REGION Network 1
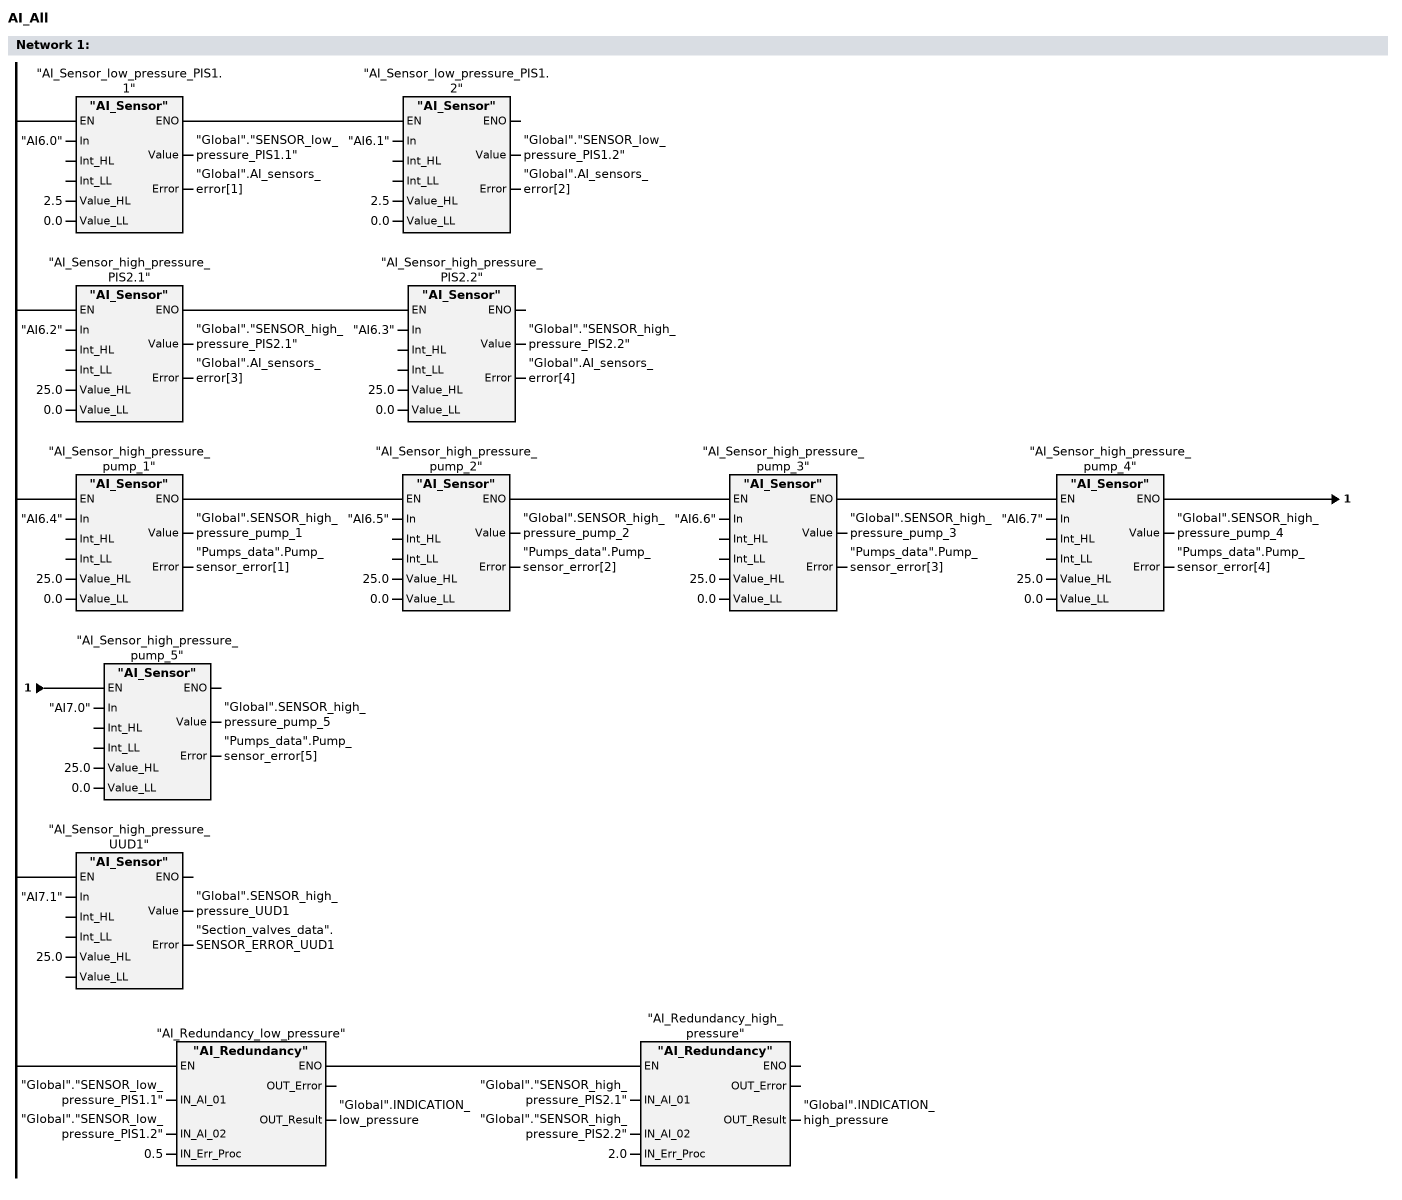
   RUNG wire#powerrail
      "AI_Sensor_low_pressure_PIS1.1"(In := "AI6.0", Int_HL :=, Int_LL :=, Value_HL := 2.5, Value_LL := 0.0, Value => "Global"."SENSOR_low_pressure_PIS1.1", Error => "Global".AI_sensors_error[1])
      "AI_Sensor_low_pressure_PIS1.2"(In := "AI6.1", Int_HL :=, Int_LL :=, Value_HL := 2.5, Value_LL := 0.0, Value => "Global"."SENSOR_low_pressure_PIS1.2", Error => "Global".AI_sensors_error[2])
   END_RUNG
   RUNG wire#powerrail
      "AI_Sensor_high_pressure_PIS2.1"(In := "AI6.2", Int_HL :=, Int_LL :=, Value_HL := 25.0, Value_LL := 0.0, Value => "Global"."SENSOR_high_pressure_PIS2.1", Error => "Global".AI_sensors_error[3])
      "AI_Sensor_high_pressure_PIS2.2"(In := "AI6.3", Int_HL :=, Int_LL :=, Value_HL := 25.0, Value_LL := 0.0, Value => "Global"."SENSOR_high_pressure_PIS2.2", Error => "Global".AI_sensors_error[4])
   END_RUNG
   RUNG wire#powerrail
      "AI_Sensor_high_pressure_pump_1"(In := "AI6.4", Int_HL :=, Int_LL :=, Value_HL := 25.0, Value_LL := 0.0, Value => "Global".SENSOR_high_pressure_pump_1, Error => "Pumps_data".Pump_sensor_error[1])
      "AI_Sensor_high_pressure_pump_2"(In := "AI6.5", Int_HL :=, Int_LL :=, Value_HL := 25.0, Value_LL := 0.0, Value => "Global".SENSOR_high_pressure_pump_2, Error => "Pumps_data".Pump_sensor_error[2])
      "AI_Sensor_high_pressure_pump_3"(In := "AI6.6", Int_HL :=, Int_LL :=, Value_HL := 25.0, Value_LL := 0.0, Value => "Global".SENSOR_high_pressure_pump_3, Error => "Pumps_data".Pump_sensor_error[3])
      "AI_Sensor_high_pressure_pump_4"(In := "AI6.7", Int_HL :=, Int_LL :=, Value_HL := 25.0, Value_LL := 0.0, Value => "Global".SENSOR_high_pressure_pump_4, Error => "Pumps_data".Pump_sensor_error[4])
      "AI_Sensor_high_pressure_pump_5"(In := "AI7.0", Int_HL :=, Int_LL :=, Value_HL := 25.0, Value_LL := 0.0, Value => "Global".SENSOR_high_pressure_pump_5, Error => "Pumps_data".Pump_sensor_error[5])
   END_RUNG
   RUNG wire#powerrail
      "AI_Sensor_high_pressure_UUD1"(In := "AI7.1", Int_HL :=, Int_LL :=, Value_HL := 25.0, Value_LL :=, Value => "Global".SENSOR_high_pressure_UUD1, Error => "Section_valves_data".SENSOR_ERROR_UUD1)
   END_RUNG
   RUNG wire#powerrail
      "AI_Redundancy_low_pressure"(IN_AI_01 := "Global"."SENSOR_low_pressure_PIS1.1", IN_AI_02 := "Global"."SENSOR_low_pressure_PIS1.2", IN_Err_Proc := 0.5, OUT_Error =>, OUT_Result => "Global".INDICATION_low_pressure)
      "AI_Redundancy_high_pressure"(IN_AI_01 := "Global"."SENSOR_high_pressure_PIS2.1", IN_AI_02 := "Global"."SENSOR_high_pressure_PIS2.2", IN_Err_Proc := 2.0, OUT_Error =>, OUT_Result => "Global".INDICATION_high_pressure)
   END_RUNG
   // the same network as SCL:
   "AI_Sensor_low_pressure_PIS1.1"(In := "AI6.0",   // "AI_Sensor"
                           Value_HL := 2.5,
                           Value_LL := 0.0,
                           Value => "Global"."SENSOR_low_pressure_PIS1.1",
                           Error => "Global".AI_sensors_error[1],
                           ENO => #_w1);
   IF #_w1 THEN
       "AI_Sensor_low_pressure_PIS1.2"(In := "AI6.1",   // "AI_Sensor"
                               Value_HL := 2.5,
                               Value_LL := 0.0,
                               Value => "Global"."SENSOR_low_pressure_PIS1.2",
                               Error => "Global".AI_sensors_error[2]);
   END_IF;
   "AI_Sensor_high_pressure_PIS2.1"(In := "AI6.2",   // "AI_Sensor"
                           Value_HL := 25.0,
                           Value_LL := 0.0,
                           Value => "Global"."SENSOR_high_pressure_PIS2.1",
                           Error => "Global".AI_sensors_error[3],
                           ENO => #_w2);
   IF #_w2 THEN
       "AI_Sensor_high_pressure_PIS2.2"(In := "AI6.3",   // "AI_Sensor"
                               Value_HL := 25.0,
                               Value_LL := 0.0,
                               Value => "Global"."SENSOR_high_pressure_PIS2.2",
                               Error => "Global".AI_sensors_error[4]);
   END_IF;
   "AI_Sensor_high_pressure_pump_1"(In := "AI6.4",   // "AI_Sensor"
                           Value_HL := 25.0,
                           Value_LL := 0.0,
                           Value => "Global".SENSOR_high_pressure_pump_1,
                           Error => "Pumps_data".Pump_sensor_error[1],
                           ENO => #_w3);
   "AI_Sensor_high_pressure_pump_2"(EN := #_w3,   // "AI_Sensor"
                           In := "AI6.5",
                           Value_HL := 25.0,
                           Value_LL := 0.0,
                           Value => "Global".SENSOR_high_pressure_pump_2,
                           Error => "Pumps_data".Pump_sensor_error[2],
                           ENO => #_w4);
   "AI_Sensor_high_pressure_pump_3"(EN := #_w4,   // "AI_Sensor"
                           In := "AI6.6",
                           Value_HL := 25.0,
                           Value_LL := 0.0,
                           Value => "Global".SENSOR_high_pressure_pump_3,
                           Error => "Pumps_data".Pump_sensor_error[3],
                           ENO => #_w5);
   "AI_Sensor_high_pressure_pump_4"(EN := #_w5,   // "AI_Sensor"
                           In := "AI6.7",
                           Value_HL := 25.0,
                           Value_LL := 0.0,
                           Value => "Global".SENSOR_high_pressure_pump_4,
                           Error => "Pumps_data".Pump_sensor_error[4],
                           ENO => #_w6);
   IF #_w6 THEN
       "AI_Sensor_high_pressure_pump_5"(In := "AI7.0",   // "AI_Sensor"
                               Value_HL := 25.0,
                               Value_LL := 0.0,
                               Value => "Global".SENSOR_high_pressure_pump_5,
                               Error => "Pumps_data".Pump_sensor_error[5]);
   END_IF;
   "AI_Sensor_high_pressure_UUD1"(In := "AI7.1",   // "AI_Sensor"
                           Value_HL := 25.0,
                           Value => "Global".SENSOR_high_pressure_UUD1,
                           Error => "Section_valves_data".SENSOR_ERROR_UUD1);
   "AI_Redundancy_low_pressure"(IN_AI_01 := "Global"."SENSOR_low_pressure_PIS1.1",   // "AI_Redundancy"
                           IN_AI_02 := "Global"."SENSOR_low_pressure_PIS1.2",
                           IN_Err_Proc := 0.5,
                           OUT_Result => "Global".INDICATION_low_pressure,
                           ENO => #_w7);
   IF #_w7 THEN
       "AI_Redundancy_high_pressure"(IN_AI_01 := "Global"."SENSOR_high_pressure_PIS2.1",   // "AI_Redundancy"
                               IN_AI_02 := "Global"."SENSOR_high_pressure_PIS2.2",
                               IN_Err_Proc := 2.0,
                               OUT_Result => "Global".INDICATION_high_pressure);
   END_IF;
END_REGION
END_FUNCTION

ORGANIZATION_BLOCK "Main"   // OB1, LAD, ProgramCycle
TITLE = "Main Program Sweep (Cycle)"
{ S7_Optimized_Access := 'TRUE' }
VERSION : 0.1
   VAR_INPUT
      Initial_Call : Bool;   // Initial call of this OB
      Remanence : Bool;   // =True, if remanent data are available
   END_VAR
   VAR_TEMP   // added for the SCL form of the ladder/FBD networks
      _w1 : Bool;
   END_VAR
BEGIN

REGION Network 1: Обработка входов
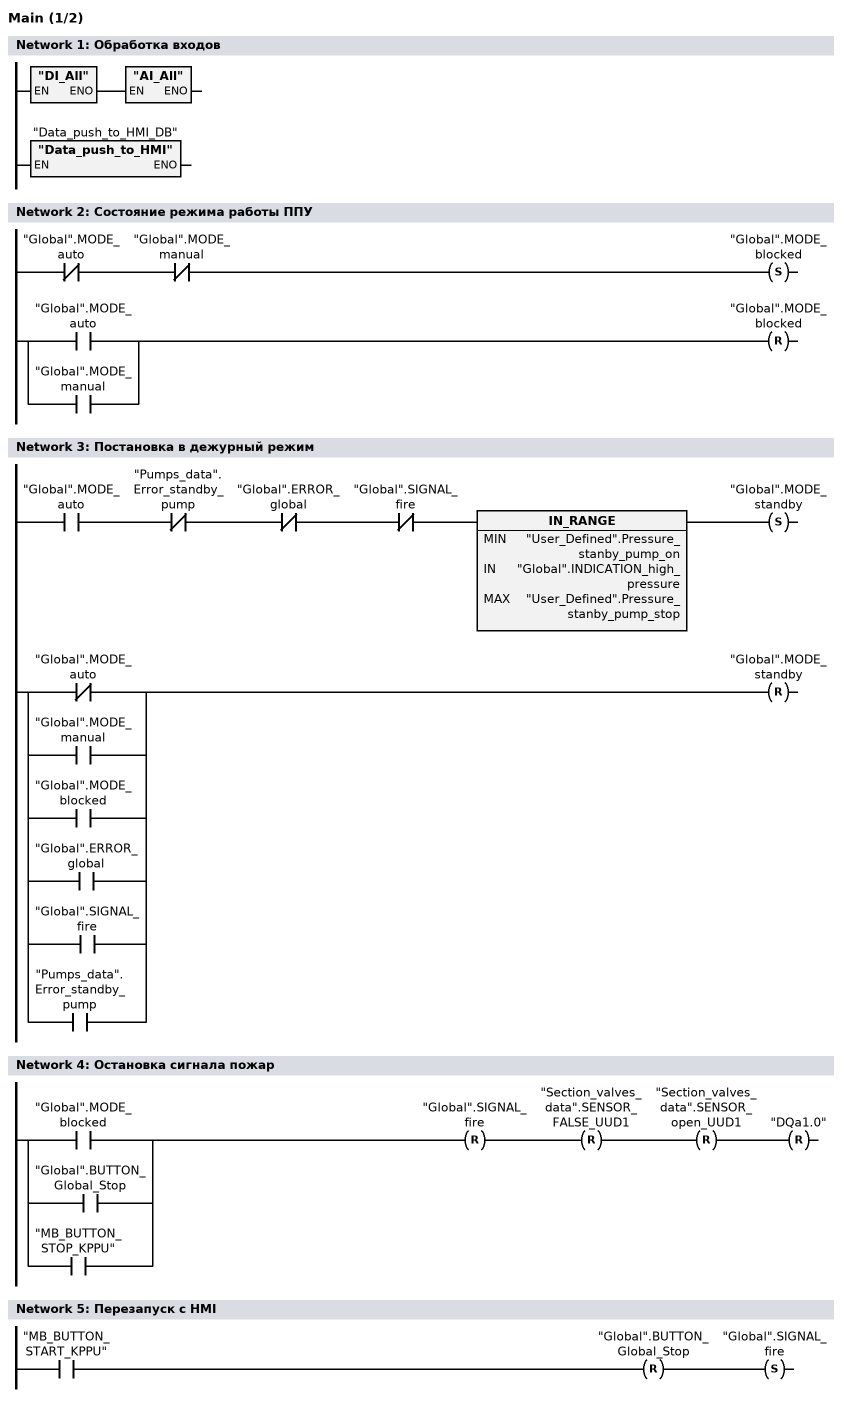
   RUNG wire#powerrail
      "DI_All"()
      "AI_All"()
   END_RUNG
   RUNG wire#powerrail
      "Data_push_to_HMI_DB"()
   END_RUNG
   // the same network as SCL:
   "DI_All"(ENO => #_w1);
   IF #_w1 THEN "AI_All"(); END_IF;
   "Data_push_to_HMI_DB"();   // "Data_push_to_HMI"
END_REGION

REGION Network 2: Состояние режима работы ППУ
   RUNG wire#powerrail
      I_Contact( "Global".MODE_auto )
      I_Contact( "Global".MODE_manual )
      S_Coil( "Global".MODE_blocked )
   END_RUNG
   RUNG wire#powerrail
      Contact( "Global".MODE_auto )
      wire#w1
      R_Coil( "Global".MODE_blocked )
   END_RUNG
   RUNG wire#powerrail
      Contact( "Global".MODE_manual )
   END_RUNG wire#w1
   // the same network as SCL:
   IF NOT "Global".MODE_auto AND NOT "Global".MODE_manual THEN "Global".MODE_blocked := TRUE; END_IF;
   IF "Global".MODE_auto OR "Global".MODE_manual THEN "Global".MODE_blocked := FALSE; END_IF;
END_REGION

REGION Network 3: Постановка в дежурный режим
   RUNG wire#powerrail
      Contact( "Global".MODE_auto )
      I_Contact( "Pumps_data".Error_standby_pump )
      I_Contact( "Global".ERROR_global )
      I_Contact( "Global".SIGNAL_fire )
      { S7_Templates := "SrcType := Real" } InRange(min := "User_Defined".Pressure_stanby_pump_on, in := "Global".INDICATION_high_pressure, max := "User_Defined".Pressure_stanby_pump_stop)
      S_Coil( "Global".MODE_standby )
   END_RUNG
   RUNG wire#powerrail
      I_Contact( "Global".MODE_auto )
      wire#w1
      R_Coil( "Global".MODE_standby )
   END_RUNG
   RUNG wire#powerrail
      Contact( "Global".MODE_manual )
   END_RUNG wire#w1
   RUNG wire#powerrail
      Contact( "Global".MODE_blocked )
   END_RUNG wire#w1
   RUNG wire#powerrail
      Contact( "Global".ERROR_global )
   END_RUNG wire#w1
   RUNG wire#powerrail
      Contact( "Global".SIGNAL_fire )
   END_RUNG wire#w1
   RUNG wire#powerrail
      Contact( "Pumps_data".Error_standby_pump )
   END_RUNG wire#w1
   // the same network as SCL:
   IF "Global".MODE_auto AND NOT "Pumps_data".Error_standby_pump AND NOT "Global".ERROR_global AND NOT "Global".SIGNAL_fire AND ("User_Defined".Pressure_stanby_pump_on <= "Global".INDICATION_high_pressure) AND ("Global".INDICATION_high_pressure <= "User_Defined".Pressure_stanby_pump_stop) THEN
       "Global".MODE_standby := TRUE;
   END_IF;
   IF NOT "Global".MODE_auto OR "Global".MODE_manual OR "Global".MODE_blocked OR "Global".ERROR_global OR "Global".SIGNAL_fire OR "Pumps_data".Error_standby_pump THEN
       "Global".MODE_standby := FALSE;
   END_IF;
END_REGION

REGION Network 4: Остановка сигнала пожар
   RUNG wire#powerrail
      Contact( "Global".MODE_blocked )
      wire#w1
      R_Coil( "Global".SIGNAL_fire )
      R_Coil( "Section_valves_data".SENSOR_FALSE_UUD1 )
      R_Coil( "Section_valves_data".SENSOR_open_UUD1 )
      R_Coil( "DQa1.0" )
   END_RUNG
   RUNG wire#powerrail
      Contact( "Global".BUTTON_Global_Stop )
   END_RUNG wire#w1
   RUNG wire#powerrail
      Contact( "MB_BUTTON_STOP_KPPU" )
   END_RUNG wire#w1
   // the same network as SCL:
   IF "Global".MODE_blocked OR "Global".BUTTON_Global_Stop OR "MB_BUTTON_STOP_KPPU" THEN
       "Global".SIGNAL_fire := FALSE;
       "Section_valves_data".SENSOR_FALSE_UUD1 := FALSE;
       "Section_valves_data".SENSOR_open_UUD1 := FALSE;
       "DQa1.0" := FALSE;
   END_IF;
END_REGION

REGION Network 5: Перезапуск с HMI
   RUNG wire#powerrail
      Contact( "MB_BUTTON_START_KPPU" )
      R_Coil( "Global".BUTTON_Global_Stop )
      S_Coil( "Global".SIGNAL_fire )
   END_RUNG
   // the same network as SCL:
   IF "MB_BUTTON_START_KPPU" THEN
       "Global".BUTTON_Global_Stop := FALSE;
       "Global".SIGNAL_fire := TRUE;
   END_IF;
END_REGION

REGION Network 6
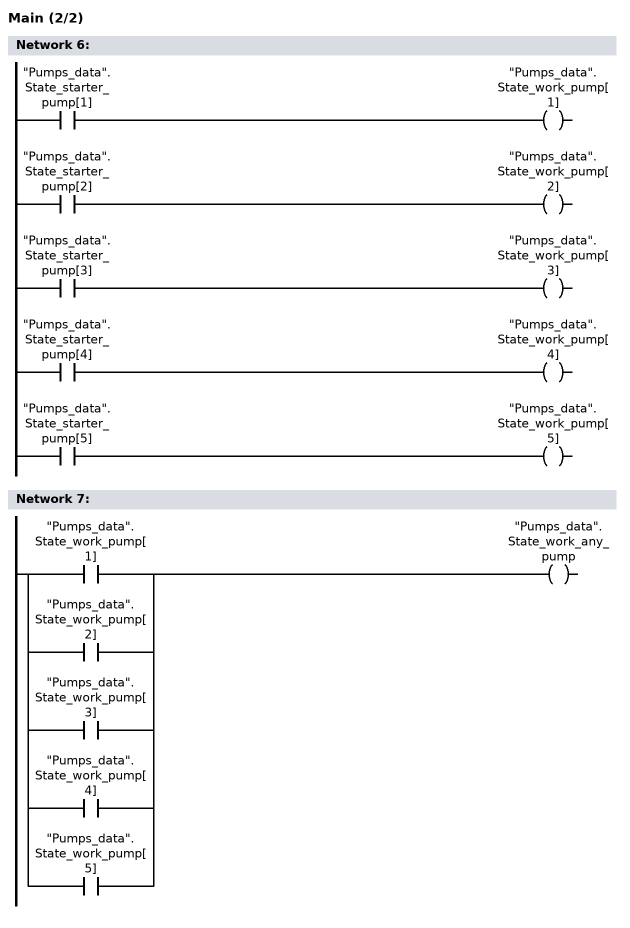
   RUNG wire#powerrail
      Contact( "Pumps_data".State_starter_pump[1] )
      Coil( "Pumps_data".State_work_pump[1] )
   END_RUNG
   RUNG wire#powerrail
      Contact( "Pumps_data".State_starter_pump[2] )
      Coil( "Pumps_data".State_work_pump[2] )
   END_RUNG
   RUNG wire#powerrail
      Contact( "Pumps_data".State_starter_pump[3] )
      Coil( "Pumps_data".State_work_pump[3] )
   END_RUNG
   RUNG wire#powerrail
      Contact( "Pumps_data".State_starter_pump[4] )
      Coil( "Pumps_data".State_work_pump[4] )
   END_RUNG
   RUNG wire#powerrail
      Contact( "Pumps_data".State_starter_pump[5] )
      Coil( "Pumps_data".State_work_pump[5] )
   END_RUNG
   // the same network as SCL:
   "Pumps_data".State_work_pump[1] := "Pumps_data".State_starter_pump[1];
   "Pumps_data".State_work_pump[2] := "Pumps_data".State_starter_pump[2];
   "Pumps_data".State_work_pump[3] := "Pumps_data".State_starter_pump[3];
   "Pumps_data".State_work_pump[4] := "Pumps_data".State_starter_pump[4];
   "Pumps_data".State_work_pump[5] := "Pumps_data".State_starter_pump[5];
END_REGION

REGION Network 7
   RUNG wire#powerrail
      Contact( "Pumps_data".State_work_pump[1] )
      wire#w1
      Coil( "Pumps_data".State_work_any_pump )
   END_RUNG
   RUNG wire#powerrail
      Contact( "Pumps_data".State_work_pump[2] )
   END_RUNG wire#w1
   RUNG wire#powerrail
      Contact( "Pumps_data".State_work_pump[3] )
   END_RUNG wire#w1
   RUNG wire#powerrail
      Contact( "Pumps_data".State_work_pump[4] )
   END_RUNG wire#w1
   RUNG wire#powerrail
      Contact( "Pumps_data".State_work_pump[5] )
   END_RUNG wire#w1
   // the same network as SCL:
   "Pumps_data".State_work_any_pump := "Pumps_data".State_work_pump[1] OR "Pumps_data".State_work_pump[2] OR "Pumps_data".State_work_pump[3] OR "Pumps_data".State_work_pump[4] OR "Pumps_data".State_work_pump[5];
END_REGION
END_ORGANIZATION_BLOCK

ORGANIZATION_BLOCK "Buttons"   // OB123, LAD, ProgramCycle
TITLE = "Main Program Sweep (Cycle)"
{ S7_Optimized_Access := 'TRUE' }
VERSION : 0.1
   VAR_INPUT
      Initial_Call : Bool;   // Initial call of this OB
      Remanence : Bool;   // =True, if remanent data are available
   END_VAR
   VAR_TEMP   // added for the SCL form of the ladder/FBD networks
      _w1 : Bool;
   END_VAR
BEGIN

REGION Network 1: Кнопка СТОП
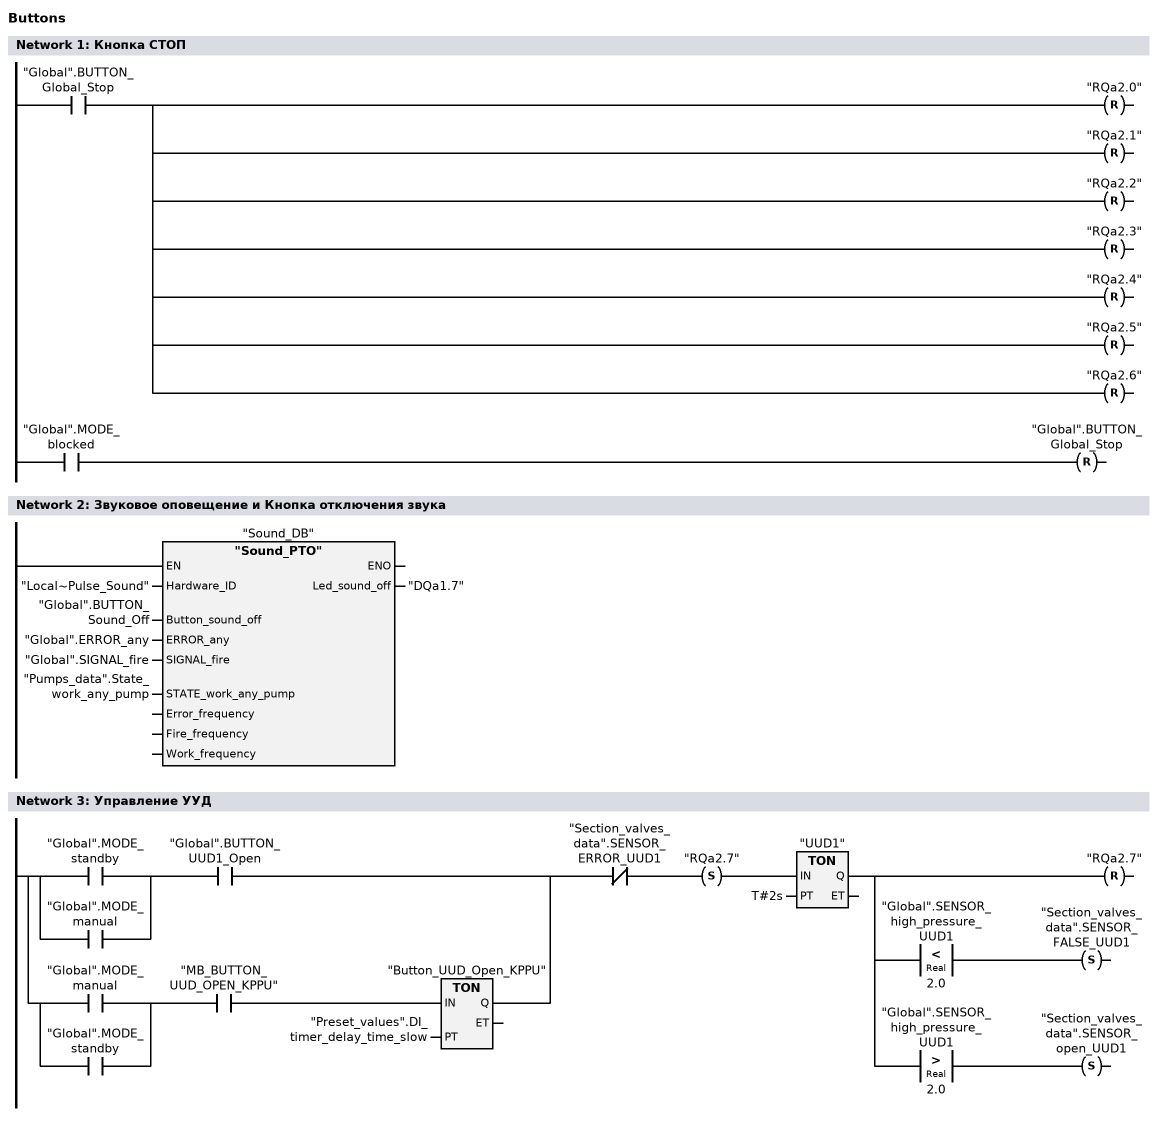
   RUNG wire#powerrail
      Contact( "Global".BUTTON_Global_Stop )
      wire#w1
      R_Coil( "RQa2.0" )
   END_RUNG
   RUNG wire#w1
      R_Coil( "RQa2.1" )
   END_RUNG
   RUNG wire#w1
      R_Coil( "RQa2.2" )
   END_RUNG
   RUNG wire#w1
      R_Coil( "RQa2.3" )
   END_RUNG
   RUNG wire#w1
      R_Coil( "RQa2.4" )
   END_RUNG
   RUNG wire#w1
      R_Coil( "RQa2.5" )
   END_RUNG
   RUNG wire#w1
      R_Coil( "RQa2.6" )
   END_RUNG
   RUNG wire#powerrail
      Contact( "Global".MODE_blocked )
      R_Coil( "Global".BUTTON_Global_Stop )
   END_RUNG
   // the same network as SCL:
   IF "Global".BUTTON_Global_Stop THEN
       "RQa2.0" := FALSE;
       "RQa2.1" := FALSE;
       "RQa2.2" := FALSE;
       "RQa2.3" := FALSE;
       "RQa2.4" := FALSE;
       "RQa2.5" := FALSE;
       "RQa2.6" := FALSE;
   END_IF;
   IF "Global".MODE_blocked THEN "Global".BUTTON_Global_Stop := FALSE; END_IF;
END_REGION

REGION Network 2: Звуковое оповещение и Кнопка отключения звука
   RUNG wire#powerrail
      "Sound_DB"(Hardware_ID := "Local~Pulse_Sound", Button_sound_off := "Global".BUTTON_Sound_Off, ERROR_any := "Global".ERROR_any, SIGNAL_fire := "Global".SIGNAL_fire, STATE_work_any_pump := "Pumps_data".State_work_any_pump, Error_frequency :=, Fire_frequency :=, Work_frequency :=, Led_sound_off => "DQa1.7")
   END_RUNG
   // the same network as SCL:
   "Sound_DB"(Hardware_ID := "Local~Pulse_Sound",   // "Sound_PTO"
              Button_sound_off := "Global".BUTTON_Sound_Off,
              ERROR_any := "Global".ERROR_any,
              SIGNAL_fire := "Global".SIGNAL_fire,
              STATE_work_any_pump := "Pumps_data".State_work_any_pump,
              Led_sound_off => "DQa1.7");
END_REGION

REGION Network 3: Управление УУД
   "Button_UUD_Open_KPPU".TON(IN := ("Global".MODE_manual OR "Global".MODE_standby) AND "MB_BUTTON_UUD_OPEN_KPPU",
                           PT := "Preset_values".DI_timer_delay_time_slow);
   #_w1 := ((("Global".MODE_standby OR "Global".MODE_manual) AND "Global".BUTTON_UUD1_Open) OR "Button_UUD_Open_KPPU".Q) AND NOT "Section_valves_data".SENSOR_ERROR_UUD1;
   IF #_w1 THEN "RQa2.7" := TRUE; END_IF;
   "UUD1".TON(IN := #_w1, PT := T#2s);
   IF "UUD1".Q THEN "RQa2.7" := FALSE; END_IF;
   IF "UUD1".Q AND ("Global".SENSOR_high_pressure_UUD1 < 2.0) THEN
       "Section_valves_data".SENSOR_FALSE_UUD1 := TRUE;
   END_IF;
   IF "UUD1".Q AND ("Global".SENSOR_high_pressure_UUD1 > 2.0) THEN
       "Section_valves_data".SENSOR_open_UUD1 := TRUE;
   END_IF;
END_REGION
END_ORGANIZATION_BLOCK

ORGANIZATION_BLOCK "Errors"   // OB124, LAD, ProgramCycle
TITLE = "Main Program Sweep (Cycle)"
{ S7_Optimized_Access := 'TRUE' }
VERSION : 0.1
   VAR_INPUT
      Initial_Call : Bool;   // Initial call of this OB
      Remanence : Bool;   // =True, if remanent data are available
   END_VAR
   VAR_TEMP   // added for the SCL form of the ladder/FBD networks
      _w1 : Bool;
      _w2 : Bool;
      _w3 : Bool;
      _w4 : Bool;
   END_VAR
BEGIN

REGION Network 1: Нет воды
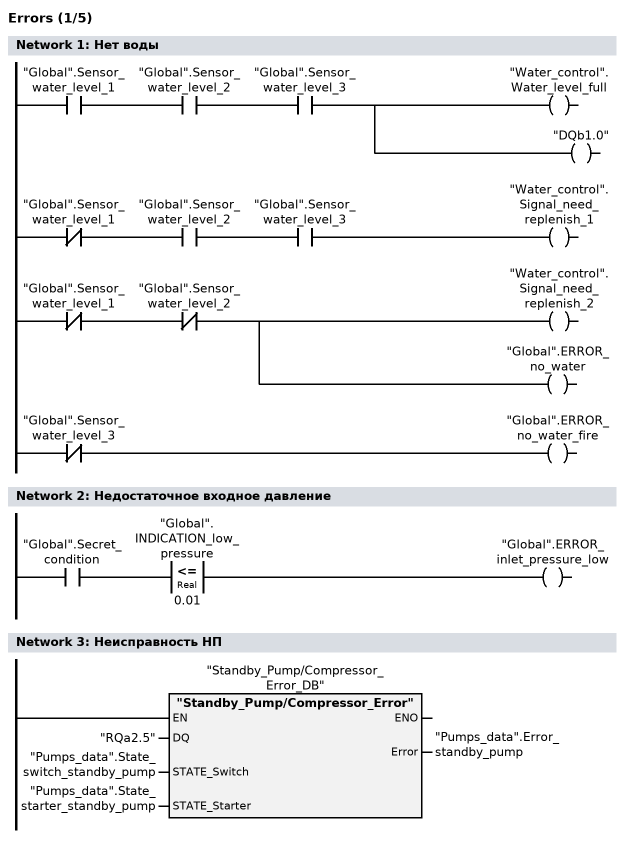
   RUNG wire#powerrail
      Contact( "Global".Sensor_water_level_1 )
      Contact( "Global".Sensor_water_level_2 )
      Contact( "Global".Sensor_water_level_3 )
      wire#w1
      Coil( "Water_control".Water_level_full )
   END_RUNG
   RUNG wire#w1
      Coil( "DQb1.0" )
   END_RUNG
   RUNG wire#powerrail
      I_Contact( "Global".Sensor_water_level_1 )
      Contact( "Global".Sensor_water_level_2 )
      Contact( "Global".Sensor_water_level_3 )
      Coil( "Water_control".Signal_need_replenish_1 )
   END_RUNG
   RUNG wire#powerrail
      I_Contact( "Global".Sensor_water_level_1 )
      I_Contact( "Global".Sensor_water_level_2 )
      wire#w2
      Coil( "Water_control".Signal_need_replenish_2 )
   END_RUNG
   RUNG wire#w2
      Coil( "Global".ERROR_no_water )
   END_RUNG
   RUNG wire#powerrail
      I_Contact( "Global".Sensor_water_level_3 )
      Coil( "Global".ERROR_no_water_fire )
   END_RUNG
   // the same network as SCL:
   "Water_control".Water_level_full := "Global".Sensor_water_level_1 AND "Global".Sensor_water_level_2 AND "Global".Sensor_water_level_3;
   "DQb1.0" := "Water_control".Water_level_full;
   "Water_control".Signal_need_replenish_1 := NOT "Global".Sensor_water_level_1 AND "Global".Sensor_water_level_2 AND "Global".Sensor_water_level_3;
   "Water_control".Signal_need_replenish_2 := NOT "Global".Sensor_water_level_1 AND NOT "Global".Sensor_water_level_2;
   "Global".ERROR_no_water := "Water_control".Signal_need_replenish_2;
   "Global".ERROR_no_water_fire := NOT "Global".Sensor_water_level_3;
END_REGION

REGION Network 2: Недостаточное входное давление
   RUNG wire#powerrail
      Contact( "Global".Secret_condition )
      { S7_Templates := "SrcType := Real" } LE_Contact(in1 := "Global".INDICATION_low_pressure, in2 := 0.01)
      Coil( "Global".ERROR_inlet_pressure_low )
   END_RUNG
   // the same network as SCL:
   "Global".ERROR_inlet_pressure_low := "Global".Secret_condition AND ("Global".INDICATION_low_pressure <= 0.01);
END_REGION

REGION Network 3: Неисправность НП
   RUNG wire#powerrail
      "Standby_Pump/Compressor_Error_DB"(DQ := "RQa2.5", STATE_Switch := "Pumps_data".State_switch_standby_pump, STATE_Starter := "Pumps_data".State_starter_standby_pump, Error => "Pumps_data".Error_standby_pump)
   END_RUNG
   // the same network as SCL:
   "Standby_Pump/Compressor_Error_DB"(DQ := "RQa2.5",   // "Standby_Pump/Compressor_Error"
                           STATE_Switch := "Pumps_data".State_switch_standby_pump,
                           STATE_Starter := "Pumps_data".State_starter_standby_pump,
                           Error => "Pumps_data".Error_standby_pump);
END_REGION

REGION Network 4: Неисправности НБ
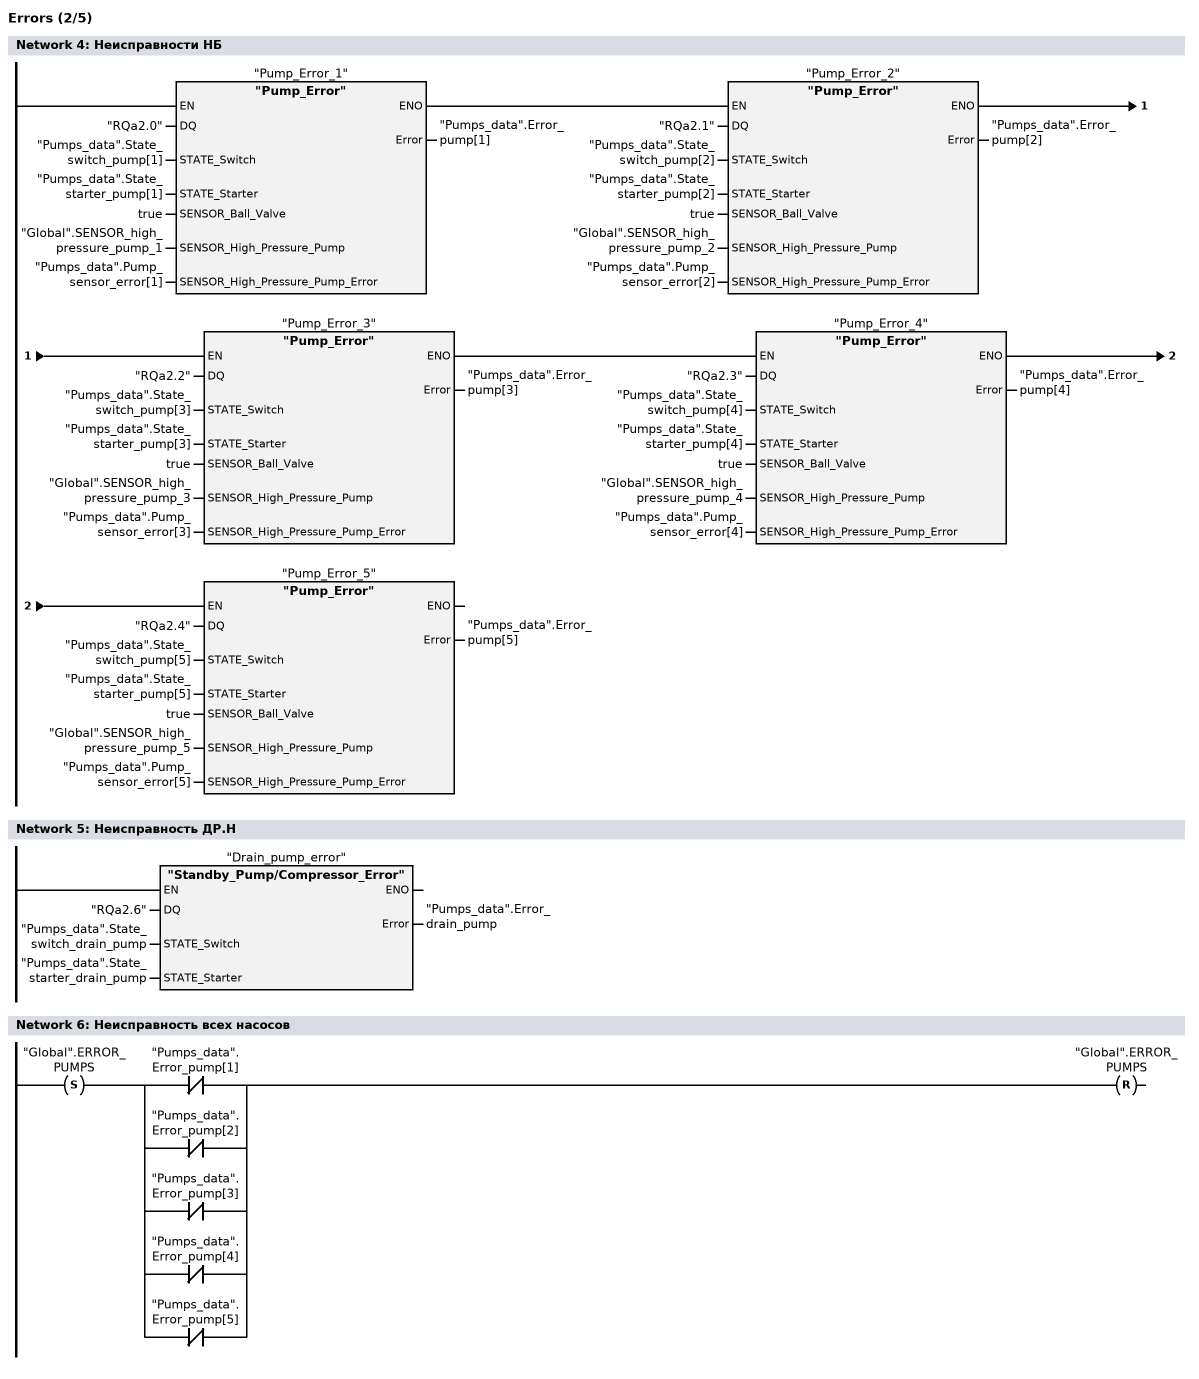
   RUNG wire#powerrail
      "Pump_Error_1"(DQ := "RQa2.0", STATE_Switch := "Pumps_data".State_switch_pump[1], STATE_Starter := "Pumps_data".State_starter_pump[1], SENSOR_Ball_Valve := true, SENSOR_High_Pressure_Pump := "Global".SENSOR_high_pressure_pump_1, SENSOR_High_Pressure_Pump_Error := "Pumps_data".Pump_sensor_error[1], Error => "Pumps_data".Error_pump[1])
      "Pump_Error_2"(DQ := "RQa2.1", STATE_Switch := "Pumps_data".State_switch_pump[2], STATE_Starter := "Pumps_data".State_starter_pump[2], SENSOR_Ball_Valve := true, SENSOR_High_Pressure_Pump := "Global".SENSOR_high_pressure_pump_2, SENSOR_High_Pressure_Pump_Error := "Pumps_data".Pump_sensor_error[2], Error => "Pumps_data".Error_pump[2])
      "Pump_Error_3"(DQ := "RQa2.2", STATE_Switch := "Pumps_data".State_switch_pump[3], STATE_Starter := "Pumps_data".State_starter_pump[3], SENSOR_Ball_Valve := true, SENSOR_High_Pressure_Pump := "Global".SENSOR_high_pressure_pump_3, SENSOR_High_Pressure_Pump_Error := "Pumps_data".Pump_sensor_error[3], Error => "Pumps_data".Error_pump[3])
      "Pump_Error_4"(DQ := "RQa2.3", STATE_Switch := "Pumps_data".State_switch_pump[4], STATE_Starter := "Pumps_data".State_starter_pump[4], SENSOR_Ball_Valve := true, SENSOR_High_Pressure_Pump := "Global".SENSOR_high_pressure_pump_4, SENSOR_High_Pressure_Pump_Error := "Pumps_data".Pump_sensor_error[4], Error => "Pumps_data".Error_pump[4])
      "Pump_Error_5"(DQ := "RQa2.4", STATE_Switch := "Pumps_data".State_switch_pump[5], STATE_Starter := "Pumps_data".State_starter_pump[5], SENSOR_Ball_Valve := true, SENSOR_High_Pressure_Pump := "Global".SENSOR_high_pressure_pump_5, SENSOR_High_Pressure_Pump_Error := "Pumps_data".Pump_sensor_error[5], Error => "Pumps_data".Error_pump[5])
   END_RUNG
   // the same network as SCL:
   "Pump_Error_1"(DQ := "RQa2.0",   // "Pump_Error"
                  STATE_Switch := "Pumps_data".State_switch_pump[1],
                  STATE_Starter := "Pumps_data".State_starter_pump[1],
                  SENSOR_Ball_Valve := true,
                  SENSOR_High_Pressure_Pump := "Global".SENSOR_high_pressure_pump_1,
                  SENSOR_High_Pressure_Pump_Error := "Pumps_data".Pump_sensor_error[1],
                  Error => "Pumps_data".Error_pump[1],
                  ENO => #_w1);
   "Pump_Error_2"(EN := #_w1,   // "Pump_Error"
                  DQ := "RQa2.1",
                  STATE_Switch := "Pumps_data".State_switch_pump[2],
                  STATE_Starter := "Pumps_data".State_starter_pump[2],
                  SENSOR_Ball_Valve := true,
                  SENSOR_High_Pressure_Pump := "Global".SENSOR_high_pressure_pump_2,
                  SENSOR_High_Pressure_Pump_Error := "Pumps_data".Pump_sensor_error[2],
                  Error => "Pumps_data".Error_pump[2],
                  ENO => #_w2);
   "Pump_Error_3"(EN := #_w2,   // "Pump_Error"
                  DQ := "RQa2.2",
                  STATE_Switch := "Pumps_data".State_switch_pump[3],
                  STATE_Starter := "Pumps_data".State_starter_pump[3],
                  SENSOR_Ball_Valve := true,
                  SENSOR_High_Pressure_Pump := "Global".SENSOR_high_pressure_pump_3,
                  SENSOR_High_Pressure_Pump_Error := "Pumps_data".Pump_sensor_error[3],
                  Error => "Pumps_data".Error_pump[3],
                  ENO => #_w3);
   "Pump_Error_4"(EN := #_w3,   // "Pump_Error"
                  DQ := "RQa2.3",
                  STATE_Switch := "Pumps_data".State_switch_pump[4],
                  STATE_Starter := "Pumps_data".State_starter_pump[4],
                  SENSOR_Ball_Valve := true,
                  SENSOR_High_Pressure_Pump := "Global".SENSOR_high_pressure_pump_4,
                  SENSOR_High_Pressure_Pump_Error := "Pumps_data".Pump_sensor_error[4],
                  Error => "Pumps_data".Error_pump[4],
                  ENO => #_w4);
   IF #_w4 THEN
       "Pump_Error_5"(DQ := "RQa2.4",   // "Pump_Error"
                      STATE_Switch := "Pumps_data".State_switch_pump[5],
                      STATE_Starter := "Pumps_data".State_starter_pump[5],
                      SENSOR_Ball_Valve := true,
                      SENSOR_High_Pressure_Pump := "Global".SENSOR_high_pressure_pump_5,
                      SENSOR_High_Pressure_Pump_Error := "Pumps_data".Pump_sensor_error[5],
                      Error => "Pumps_data".Error_pump[5]);
   END_IF;
END_REGION

REGION Network 5: Неисправность ДР.Н
   RUNG wire#powerrail
      "Drain_pump_error"(DQ := "RQa2.6", STATE_Switch := "Pumps_data".State_switch_drain_pump, STATE_Starter := "Pumps_data".State_starter_drain_pump, Error => "Pumps_data".Error_drain_pump)
   END_RUNG
   // the same network as SCL:
   "Drain_pump_error"(DQ := "RQa2.6",   // "Standby_Pump/Compressor_Error"
                      STATE_Switch := "Pumps_data".State_switch_drain_pump,
                      STATE_Starter := "Pumps_data".State_starter_drain_pump,
                      Error => "Pumps_data".Error_drain_pump);
END_REGION

REGION Network 6: Неисправность всех насосов
   RUNG wire#powerrail
      S_Coil( "Global".ERROR_PUMPS )
      wire#w1
      I_Contact( "Pumps_data".Error_pump[1] )
      wire#w2
      R_Coil( "Global".ERROR_PUMPS )
   END_RUNG
   RUNG wire#w1
      I_Contact( "Pumps_data".Error_pump[2] )
   END_RUNG wire#w2
   RUNG wire#w1
      I_Contact( "Pumps_data".Error_pump[3] )
   END_RUNG wire#w2
   RUNG wire#w1
      I_Contact( "Pumps_data".Error_pump[4] )
   END_RUNG wire#w2
   RUNG wire#w1
      I_Contact( "Pumps_data".Error_pump[5] )
   END_RUNG wire#w2
   // the same network as SCL:
   "Global".ERROR_PUMPS := TRUE;
   IF NOT "Pumps_data".Error_pump[1] OR NOT "Pumps_data".Error_pump[2] OR NOT "Pumps_data".Error_pump[3] OR NOT "Pumps_data".Error_pump[4] OR NOT "Pumps_data".Error_pump[5] THEN
       "Global".ERROR_PUMPS := FALSE;
   END_IF;
END_REGION

REGION Network 7: Неисправность любого насоса кроме резервного
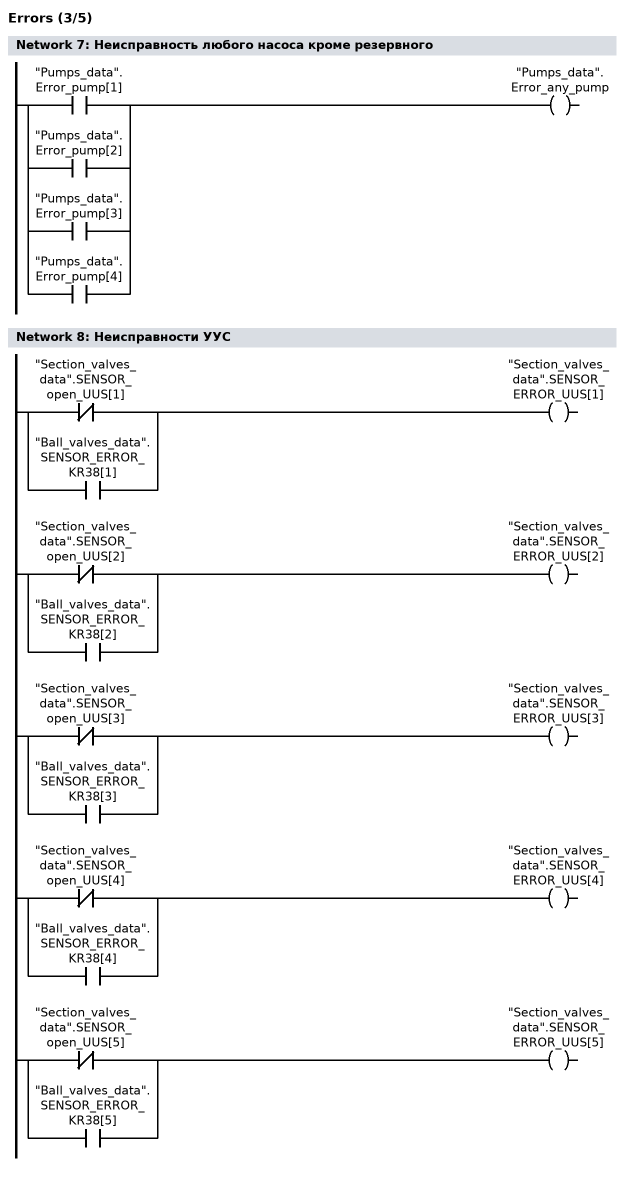
   RUNG wire#powerrail
      Contact( "Pumps_data".Error_pump[1] )
      wire#w1
      Coil( "Pumps_data".Error_any_pump )
   END_RUNG
   RUNG wire#powerrail
      Contact( "Pumps_data".Error_pump[2] )
   END_RUNG wire#w1
   RUNG wire#powerrail
      Contact( "Pumps_data".Error_pump[3] )
   END_RUNG wire#w1
   RUNG wire#powerrail
      Contact( "Pumps_data".Error_pump[4] )
   END_RUNG wire#w1
   // the same network as SCL:
   "Pumps_data".Error_any_pump := "Pumps_data".Error_pump[1] OR "Pumps_data".Error_pump[2] OR "Pumps_data".Error_pump[3] OR "Pumps_data".Error_pump[4];
END_REGION

REGION Network 8: Неисправности УУС
   RUNG wire#powerrail
      I_Contact( "Section_valves_data".SENSOR_open_UUS[1] )
      wire#w1
      Coil( "Section_valves_data".SENSOR_ERROR_UUS[1] )
   END_RUNG
   RUNG wire#powerrail
      Contact( "Ball_valves_data".SENSOR_ERROR_KR38[1] )
   END_RUNG wire#w1
   RUNG wire#powerrail
      I_Contact( "Section_valves_data".SENSOR_open_UUS[2] )
      wire#w2
      Coil( "Section_valves_data".SENSOR_ERROR_UUS[2] )
   END_RUNG
   RUNG wire#powerrail
      Contact( "Ball_valves_data".SENSOR_ERROR_KR38[2] )
   END_RUNG wire#w2
   RUNG wire#powerrail
      I_Contact( "Section_valves_data".SENSOR_open_UUS[3] )
      wire#w3
      Coil( "Section_valves_data".SENSOR_ERROR_UUS[3] )
   END_RUNG
   RUNG wire#powerrail
      Contact( "Ball_valves_data".SENSOR_ERROR_KR38[3] )
   END_RUNG wire#w3
   RUNG wire#powerrail
      I_Contact( "Section_valves_data".SENSOR_open_UUS[4] )
      wire#w4
      Coil( "Section_valves_data".SENSOR_ERROR_UUS[4] )
   END_RUNG
   RUNG wire#powerrail
      Contact( "Ball_valves_data".SENSOR_ERROR_KR38[4] )
   END_RUNG wire#w4
   RUNG wire#powerrail
      I_Contact( "Section_valves_data".SENSOR_open_UUS[5] )
      wire#w5
      Coil( "Section_valves_data".SENSOR_ERROR_UUS[5] )
   END_RUNG
   RUNG wire#powerrail
      Contact( "Ball_valves_data".SENSOR_ERROR_KR38[5] )
   END_RUNG wire#w5
   // the same network as SCL:
   "Section_valves_data".SENSOR_ERROR_UUS[1] := NOT "Section_valves_data".SENSOR_open_UUS[1] OR "Ball_valves_data".SENSOR_ERROR_KR38[1];
   "Section_valves_data".SENSOR_ERROR_UUS[2] := NOT "Section_valves_data".SENSOR_open_UUS[2] OR "Ball_valves_data".SENSOR_ERROR_KR38[2];
   "Section_valves_data".SENSOR_ERROR_UUS[3] := NOT "Section_valves_data".SENSOR_open_UUS[3] OR "Ball_valves_data".SENSOR_ERROR_KR38[3];
   "Section_valves_data".SENSOR_ERROR_UUS[4] := NOT "Section_valves_data".SENSOR_open_UUS[4] OR "Ball_valves_data".SENSOR_ERROR_KR38[4];
   "Section_valves_data".SENSOR_ERROR_UUS[5] := NOT "Section_valves_data".SENSOR_open_UUS[5] OR "Ball_valves_data".SENSOR_ERROR_KR38[5];
END_REGION

REGION Network 9: Неисправность всех УУС - все закрыты
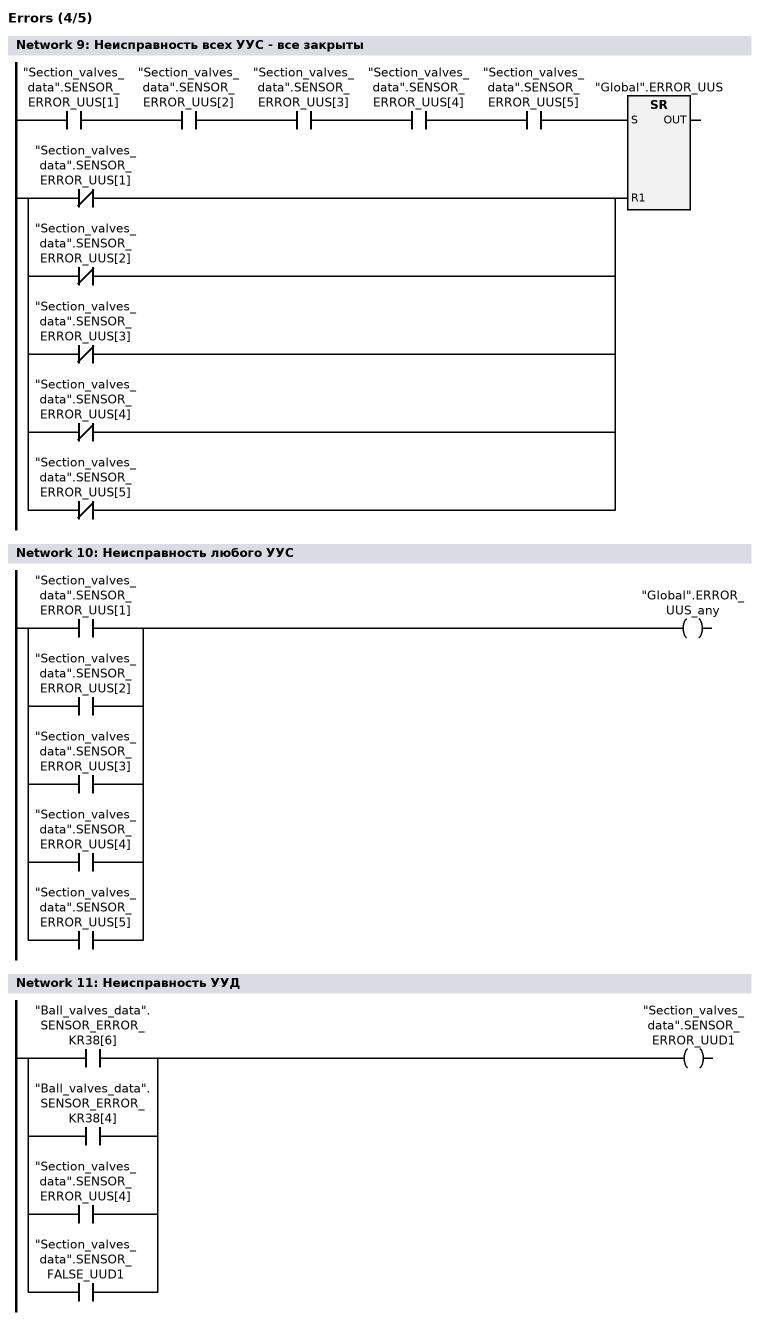
   RUNG wire#powerrail
      Contact( "Section_valves_data".SENSOR_ERROR_UUS[1] )
      Contact( "Section_valves_data".SENSOR_ERROR_UUS[2] )
      Contact( "Section_valves_data".SENSOR_ERROR_UUS[3] )
      Contact( "Section_valves_data".SENSOR_ERROR_UUS[4] )
      Contact( "Section_valves_data".SENSOR_ERROR_UUS[5] )
      S_SR(operand := "Global".ERROR_UUS, r1 := wire#w1)
   END_RUNG
   RUNG wire#powerrail
      I_Contact( "Section_valves_data".SENSOR_ERROR_UUS[1] )
   END_RUNG wire#w1
   RUNG wire#powerrail
      I_Contact( "Section_valves_data".SENSOR_ERROR_UUS[2] )
   END_RUNG wire#w1
   RUNG wire#powerrail
      I_Contact( "Section_valves_data".SENSOR_ERROR_UUS[3] )
   END_RUNG wire#w1
   RUNG wire#powerrail
      I_Contact( "Section_valves_data".SENSOR_ERROR_UUS[4] )
   END_RUNG wire#w1
   RUNG wire#powerrail
      I_Contact( "Section_valves_data".SENSOR_ERROR_UUS[5] )
   END_RUNG wire#w1
   // the same network as SCL:
   IF "Section_valves_data".SENSOR_ERROR_UUS[1] AND "Section_valves_data".SENSOR_ERROR_UUS[2] AND "Section_valves_data".SENSOR_ERROR_UUS[3] AND "Section_valves_data".SENSOR_ERROR_UUS[4] AND "Section_valves_data".SENSOR_ERROR_UUS[5] THEN
       "Global".ERROR_UUS := TRUE;   // SR flip-flop
   END_IF;
   IF NOT "Section_valves_data".SENSOR_ERROR_UUS[1] OR NOT "Section_valves_data".SENSOR_ERROR_UUS[2] OR NOT "Section_valves_data".SENSOR_ERROR_UUS[3] OR NOT "Section_valves_data".SENSOR_ERROR_UUS[4] OR NOT "Section_valves_data".SENSOR_ERROR_UUS[5] THEN
       "Global".ERROR_UUS := FALSE;
   END_IF;
END_REGION

REGION Network 10: Неисправность любого УУС
   RUNG wire#powerrail
      Contact( "Section_valves_data".SENSOR_ERROR_UUS[1] )
      wire#w1
      Coil( "Global".ERROR_UUS_any )
   END_RUNG
   RUNG wire#powerrail
      Contact( "Section_valves_data".SENSOR_ERROR_UUS[2] )
   END_RUNG wire#w1
   RUNG wire#powerrail
      Contact( "Section_valves_data".SENSOR_ERROR_UUS[3] )
   END_RUNG wire#w1
   RUNG wire#powerrail
      Contact( "Section_valves_data".SENSOR_ERROR_UUS[4] )
   END_RUNG wire#w1
   RUNG wire#powerrail
      Contact( "Section_valves_data".SENSOR_ERROR_UUS[5] )
   END_RUNG wire#w1
   // the same network as SCL:
   "Global".ERROR_UUS_any := "Section_valves_data".SENSOR_ERROR_UUS[1] OR "Section_valves_data".SENSOR_ERROR_UUS[2] OR "Section_valves_data".SENSOR_ERROR_UUS[3] OR "Section_valves_data".SENSOR_ERROR_UUS[4] OR "Section_valves_data".SENSOR_ERROR_UUS[5];
END_REGION

REGION Network 11: Неисправность УУД
   RUNG wire#powerrail
      Contact( "Ball_valves_data".SENSOR_ERROR_KR38[6] )
      wire#w1
      Coil( "Section_valves_data".SENSOR_ERROR_UUD1 )
   END_RUNG
   RUNG wire#powerrail
      Contact( "Ball_valves_data".SENSOR_ERROR_KR38[4] )
   END_RUNG wire#w1
   RUNG wire#powerrail
      Contact( "Section_valves_data".SENSOR_ERROR_UUS[4] )
   END_RUNG wire#w1
   RUNG wire#powerrail
      Contact( "Section_valves_data".SENSOR_FALSE_UUD1 )
   END_RUNG wire#w1
   // the same network as SCL:
   "Section_valves_data".SENSOR_ERROR_UUD1 := "Ball_valves_data".SENSOR_ERROR_KR38[6] OR "Ball_valves_data".SENSOR_ERROR_KR38[4] OR "Section_valves_data".SENSOR_ERROR_UUS[4] OR "Section_valves_data".SENSOR_FALSE_UUD1;
END_REGION

REGION Network 12: Неисправность любого шарового крана
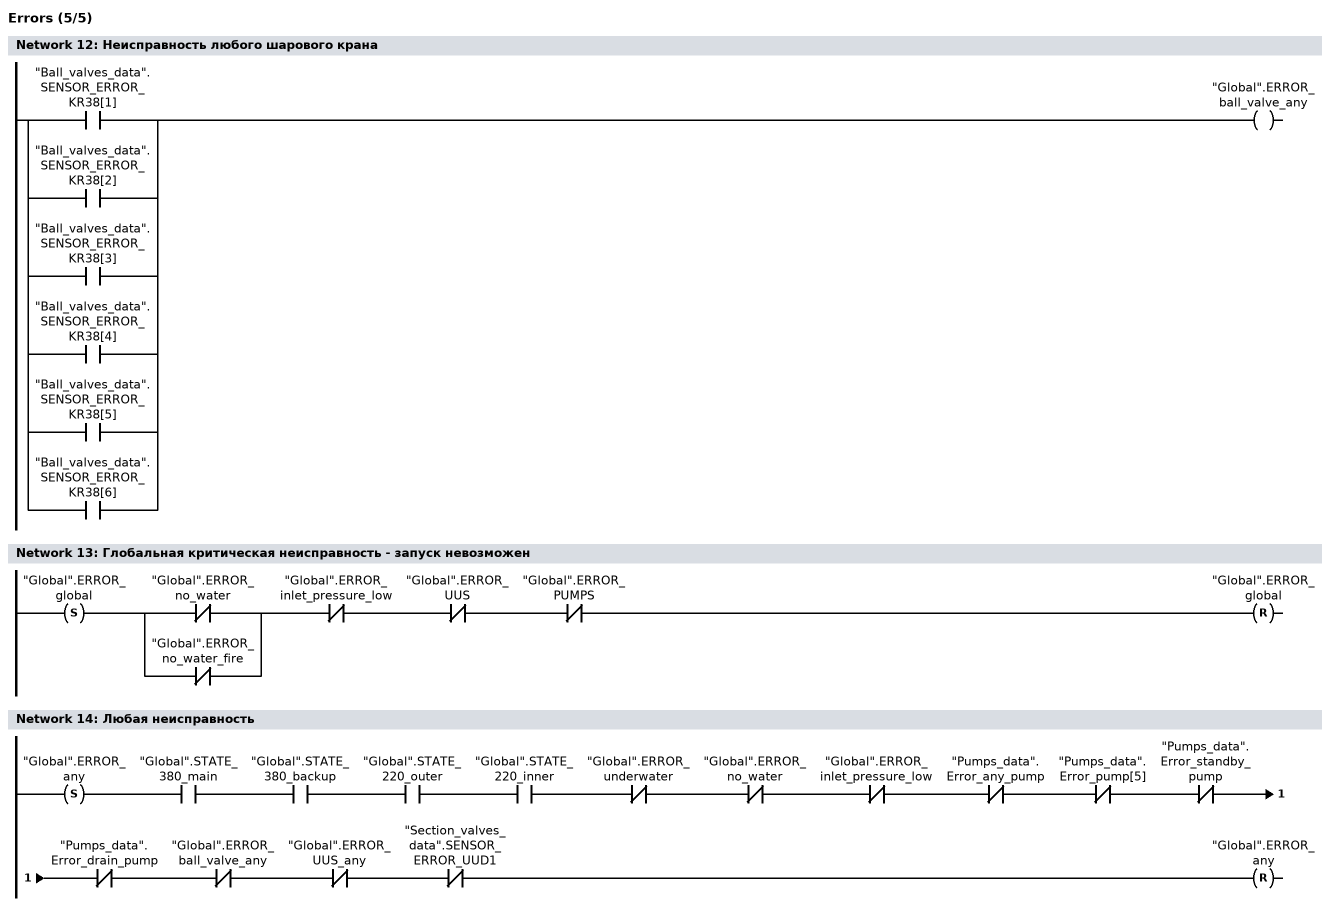
   RUNG wire#powerrail
      Contact( "Ball_valves_data".SENSOR_ERROR_KR38[1] )
      wire#w1
      Coil( "Global".ERROR_ball_valve_any )
   END_RUNG
   RUNG wire#powerrail
      Contact( "Ball_valves_data".SENSOR_ERROR_KR38[2] )
   END_RUNG wire#w1
   RUNG wire#powerrail
      Contact( "Ball_valves_data".SENSOR_ERROR_KR38[3] )
   END_RUNG wire#w1
   RUNG wire#powerrail
      Contact( "Ball_valves_data".SENSOR_ERROR_KR38[4] )
   END_RUNG wire#w1
   RUNG wire#powerrail
      Contact( "Ball_valves_data".SENSOR_ERROR_KR38[5] )
   END_RUNG wire#w1
   RUNG wire#powerrail
      Contact( "Ball_valves_data".SENSOR_ERROR_KR38[6] )
   END_RUNG wire#w1
   // the same network as SCL:
   "Global".ERROR_ball_valve_any := "Ball_valves_data".SENSOR_ERROR_KR38[1] OR "Ball_valves_data".SENSOR_ERROR_KR38[2] OR "Ball_valves_data".SENSOR_ERROR_KR38[3] OR "Ball_valves_data".SENSOR_ERROR_KR38[4] OR "Ball_valves_data".SENSOR_ERROR_KR38[5] OR "Ball_valves_data".SENSOR_ERROR_KR38[6];
END_REGION

REGION Network 13: Глобальная критическая неисправность - запуск невозможен
   RUNG wire#powerrail
      S_Coil( "Global".ERROR_global )
      wire#w1
      I_Contact( "Global".ERROR_no_water )
      wire#w2
      I_Contact( "Global".ERROR_inlet_pressure_low )
      I_Contact( "Global".ERROR_UUS )
      I_Contact( "Global".ERROR_PUMPS )
      R_Coil( "Global".ERROR_global )
   END_RUNG
   RUNG wire#w1
      I_Contact( "Global".ERROR_no_water_fire )
   END_RUNG wire#w2
   // the same network as SCL:
   "Global".ERROR_global := TRUE;
   IF (NOT "Global".ERROR_no_water OR NOT "Global".ERROR_no_water_fire) AND NOT "Global".ERROR_inlet_pressure_low AND NOT "Global".ERROR_UUS AND NOT "Global".ERROR_PUMPS THEN
       "Global".ERROR_global := FALSE;
   END_IF;
END_REGION

REGION Network 14: Любая неисправность
   RUNG wire#powerrail
      S_Coil( "Global".ERROR_any )
      Contact( "Global".STATE_380_main )
      Contact( "Global".STATE_380_backup )
      Contact( "Global".STATE_220_outer )
      Contact( "Global".STATE_220_inner )
      I_Contact( "Global".ERROR_underwater )
      I_Contact( "Global".ERROR_no_water )
      I_Contact( "Global".ERROR_inlet_pressure_low )
      I_Contact( "Pumps_data".Error_any_pump )
      I_Contact( "Pumps_data".Error_pump[5] )
      I_Contact( "Pumps_data".Error_standby_pump )
      I_Contact( "Pumps_data".Error_drain_pump )
      I_Contact( "Global".ERROR_ball_valve_any )
      I_Contact( "Global".ERROR_UUS_any )
      I_Contact( "Section_valves_data".SENSOR_ERROR_UUD1 )
      R_Coil( "Global".ERROR_any )
   END_RUNG
   // the same network as SCL:
   "Global".ERROR_any := TRUE;
   IF "Global".STATE_380_main AND "Global".STATE_380_backup AND "Global".STATE_220_outer AND "Global".STATE_220_inner AND NOT "Global".ERROR_underwater AND NOT "Global".ERROR_no_water AND NOT "Global".ERROR_inlet_pressure_low AND NOT "Pumps_data".Error_any_pump AND NOT "Pumps_data".Error_pump[5] AND NOT "Pumps_data".Error_standby_pump AND NOT "Pumps_data".Error_drain_pump AND NOT "Global".ERROR_ball_valve_any AND NOT "Global".ERROR_UUS_any AND NOT "Section_valves_data".SENSOR_ERROR_UUD1 THEN
       "Global".ERROR_any := FALSE;
   END_IF;
END_REGION
END_ORGANIZATION_BLOCK

ORGANIZATION_BLOCK "LED"   // OB125, LAD, ProgramCycle
TITLE = "Main Program Sweep (Cycle)"
{ S7_Optimized_Access := 'TRUE' }
VERSION : 0.1
   VAR_INPUT
      Initial_Call : Bool;   // Initial call of this OB
      Remanence : Bool;   // =True, if remanent data are available
   END_VAR
BEGIN

REGION Network 1: Пожар, Пуск, Неисправность, Дежурный режим, Автоматика отклчена, Система отключена
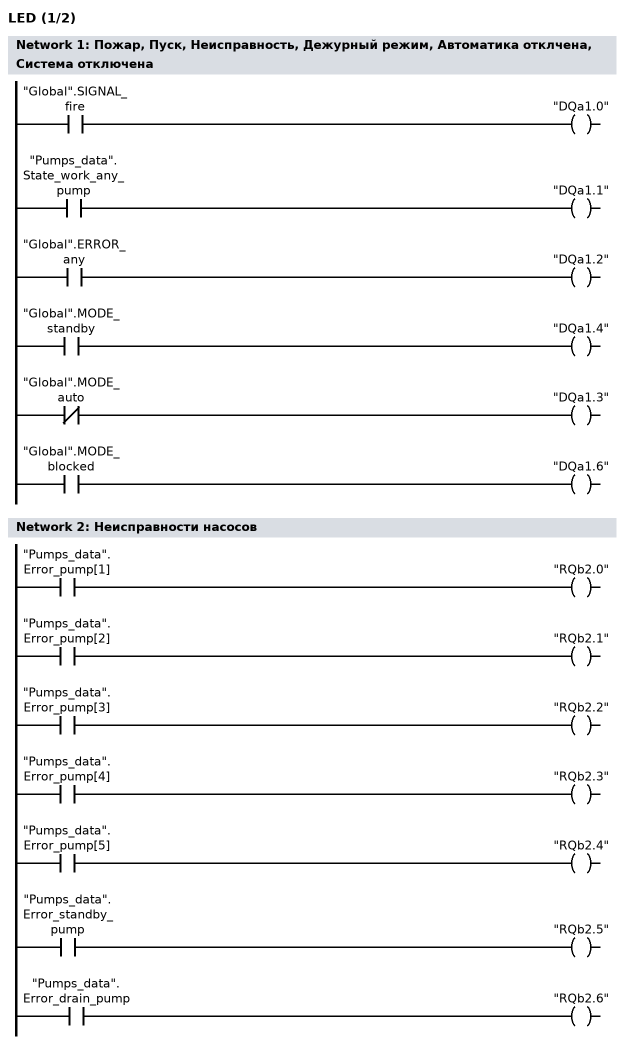
   RUNG wire#powerrail
      Contact( "Global".SIGNAL_fire )
      Coil( "DQa1.0" )
   END_RUNG
   RUNG wire#powerrail
      Contact( "Pumps_data".State_work_any_pump )
      Coil( "DQa1.1" )
   END_RUNG
   RUNG wire#powerrail
      Contact( "Global".ERROR_any )
      Coil( "DQa1.2" )
   END_RUNG
   RUNG wire#powerrail
      Contact( "Global".MODE_standby )
      Coil( "DQa1.4" )
   END_RUNG
   RUNG wire#powerrail
      I_Contact( "Global".MODE_auto )
      Coil( "DQa1.3" )
   END_RUNG
   RUNG wire#powerrail
      Contact( "Global".MODE_blocked )
      Coil( "DQa1.6" )
   END_RUNG
   // the same network as SCL:
   "DQa1.0" := "Global".SIGNAL_fire;
   "DQa1.1" := "Pumps_data".State_work_any_pump;
   "DQa1.2" := "Global".ERROR_any;
   "DQa1.4" := "Global".MODE_standby;
   "DQa1.3" := NOT "Global".MODE_auto;
   "DQa1.6" := "Global".MODE_blocked;
END_REGION

REGION Network 2: Неисправности насосов
   RUNG wire#powerrail
      Contact( "Pumps_data".Error_pump[1] )
      Coil( "RQb2.0" )
   END_RUNG
   RUNG wire#powerrail
      Contact( "Pumps_data".Error_pump[2] )
      Coil( "RQb2.1" )
   END_RUNG
   RUNG wire#powerrail
      Contact( "Pumps_data".Error_pump[3] )
      Coil( "RQb2.2" )
   END_RUNG
   RUNG wire#powerrail
      Contact( "Pumps_data".Error_pump[4] )
      Coil( "RQb2.3" )
   END_RUNG
   RUNG wire#powerrail
      Contact( "Pumps_data".Error_pump[5] )
      Coil( "RQb2.4" )
   END_RUNG
   RUNG wire#powerrail
      Contact( "Pumps_data".Error_standby_pump )
      Coil( "RQb2.5" )
   END_RUNG
   RUNG wire#powerrail
      Contact( "Pumps_data".Error_drain_pump )
      Coil( "RQb2.6" )
   END_RUNG
   // the same network as SCL:
   "RQb2.0" := "Pumps_data".Error_pump[1];
   "RQb2.1" := "Pumps_data".Error_pump[2];
   "RQb2.2" := "Pumps_data".Error_pump[3];
   "RQb2.3" := "Pumps_data".Error_pump[4];
   "RQb2.4" := "Pumps_data".Error_pump[5];
   "RQb2.5" := "Pumps_data".Error_standby_pump;
   "RQb2.6" := "Pumps_data".Error_drain_pump;
END_REGION

REGION Network 3: Неисправности УУС
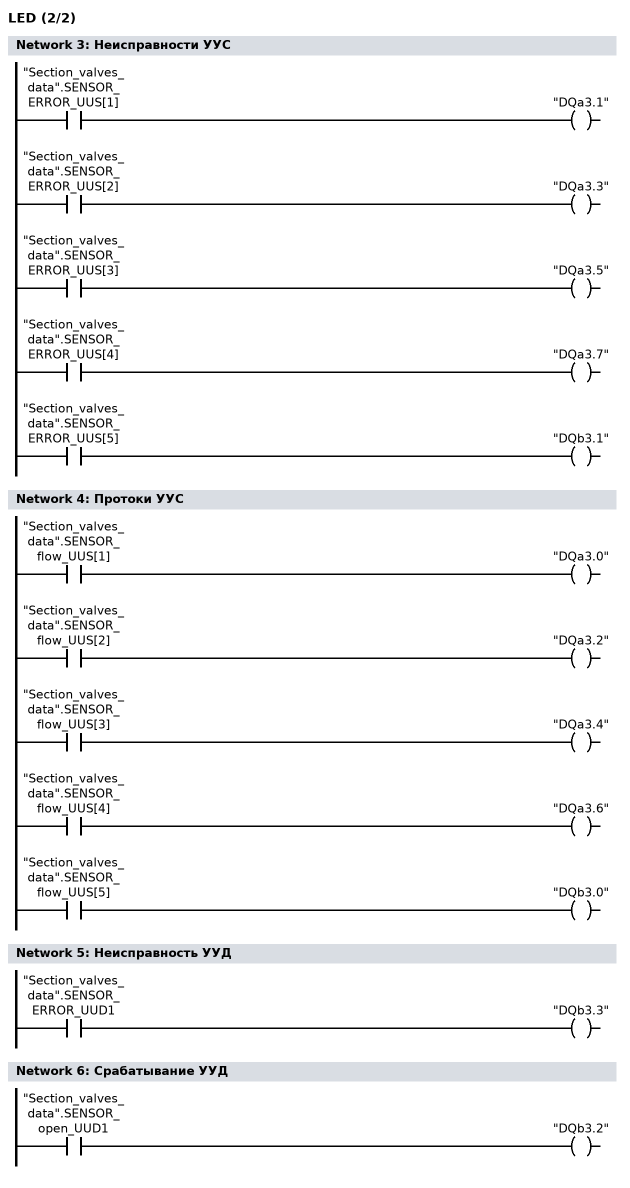
   RUNG wire#powerrail
      Contact( "Section_valves_data".SENSOR_ERROR_UUS[1] )
      Coil( "DQa3.1" )
   END_RUNG
   RUNG wire#powerrail
      Contact( "Section_valves_data".SENSOR_ERROR_UUS[2] )
      Coil( "DQa3.3" )
   END_RUNG
   RUNG wire#powerrail
      Contact( "Section_valves_data".SENSOR_ERROR_UUS[3] )
      Coil( "DQa3.5" )
   END_RUNG
   RUNG wire#powerrail
      Contact( "Section_valves_data".SENSOR_ERROR_UUS[4] )
      Coil( "DQa3.7" )
   END_RUNG
   RUNG wire#powerrail
      Contact( "Section_valves_data".SENSOR_ERROR_UUS[5] )
      Coil( "DQb3.1" )
   END_RUNG
   // the same network as SCL:
   "DQa3.1" := "Section_valves_data".SENSOR_ERROR_UUS[1];
   "DQa3.3" := "Section_valves_data".SENSOR_ERROR_UUS[2];
   "DQa3.5" := "Section_valves_data".SENSOR_ERROR_UUS[3];
   "DQa3.7" := "Section_valves_data".SENSOR_ERROR_UUS[4];
   "DQb3.1" := "Section_valves_data".SENSOR_ERROR_UUS[5];
END_REGION

REGION Network 4: Протоки УУС
   RUNG wire#powerrail
      Contact( "Section_valves_data".SENSOR_flow_UUS[1] )
      Coil( "DQa3.0" )
   END_RUNG
   RUNG wire#powerrail
      Contact( "Section_valves_data".SENSOR_flow_UUS[2] )
      Coil( "DQa3.2" )
   END_RUNG
   RUNG wire#powerrail
      Contact( "Section_valves_data".SENSOR_flow_UUS[3] )
      Coil( "DQa3.4" )
   END_RUNG
   RUNG wire#powerrail
      Contact( "Section_valves_data".SENSOR_flow_UUS[4] )
      Coil( "DQa3.6" )
   END_RUNG
   RUNG wire#powerrail
      Contact( "Section_valves_data".SENSOR_flow_UUS[5] )
      Coil( "DQb3.0" )
   END_RUNG
   // the same network as SCL:
   "DQa3.0" := "Section_valves_data".SENSOR_flow_UUS[1];
   "DQa3.2" := "Section_valves_data".SENSOR_flow_UUS[2];
   "DQa3.4" := "Section_valves_data".SENSOR_flow_UUS[3];
   "DQa3.6" := "Section_valves_data".SENSOR_flow_UUS[4];
   "DQb3.0" := "Section_valves_data".SENSOR_flow_UUS[5];
END_REGION

REGION Network 5: Неисправность УУД
   RUNG wire#powerrail
      Contact( "Section_valves_data".SENSOR_ERROR_UUD1 )
      Coil( "DQb3.3" )
   END_RUNG
   // the same network as SCL:
   "DQb3.3" := "Section_valves_data".SENSOR_ERROR_UUD1;
END_REGION

REGION Network 6: Срабатывание УУД
   RUNG wire#powerrail
      Contact( "Section_valves_data".SENSOR_open_UUD1 )
      Coil( "DQb3.2" )
   END_RUNG
   // the same network as SCL:
   "DQb3.2" := "Section_valves_data".SENSOR_open_UUD1;
END_REGION
END_ORGANIZATION_BLOCK

ORGANIZATION_BLOCK "Pumps"   // OB126, LAD, ProgramCycle
TITLE = "Main Program Sweep (Cycle)"
{ S7_Optimized_Access := 'TRUE' }
VERSION : 0.1
   VAR_INPUT
      Initial_Call : Bool;   // Initial call of this OB
      Remanence : Bool;   // =True, if remanent data are available
   END_VAR
   VAR_TEMP   // added for the SCL form of the ladder/FBD networks
      _w1 : Bool;
      _w2 : Bool;
   END_VAR
BEGIN

REGION Network 1: Работа жокей насоса и формирование сигнала ошибки давления водозаполенной части
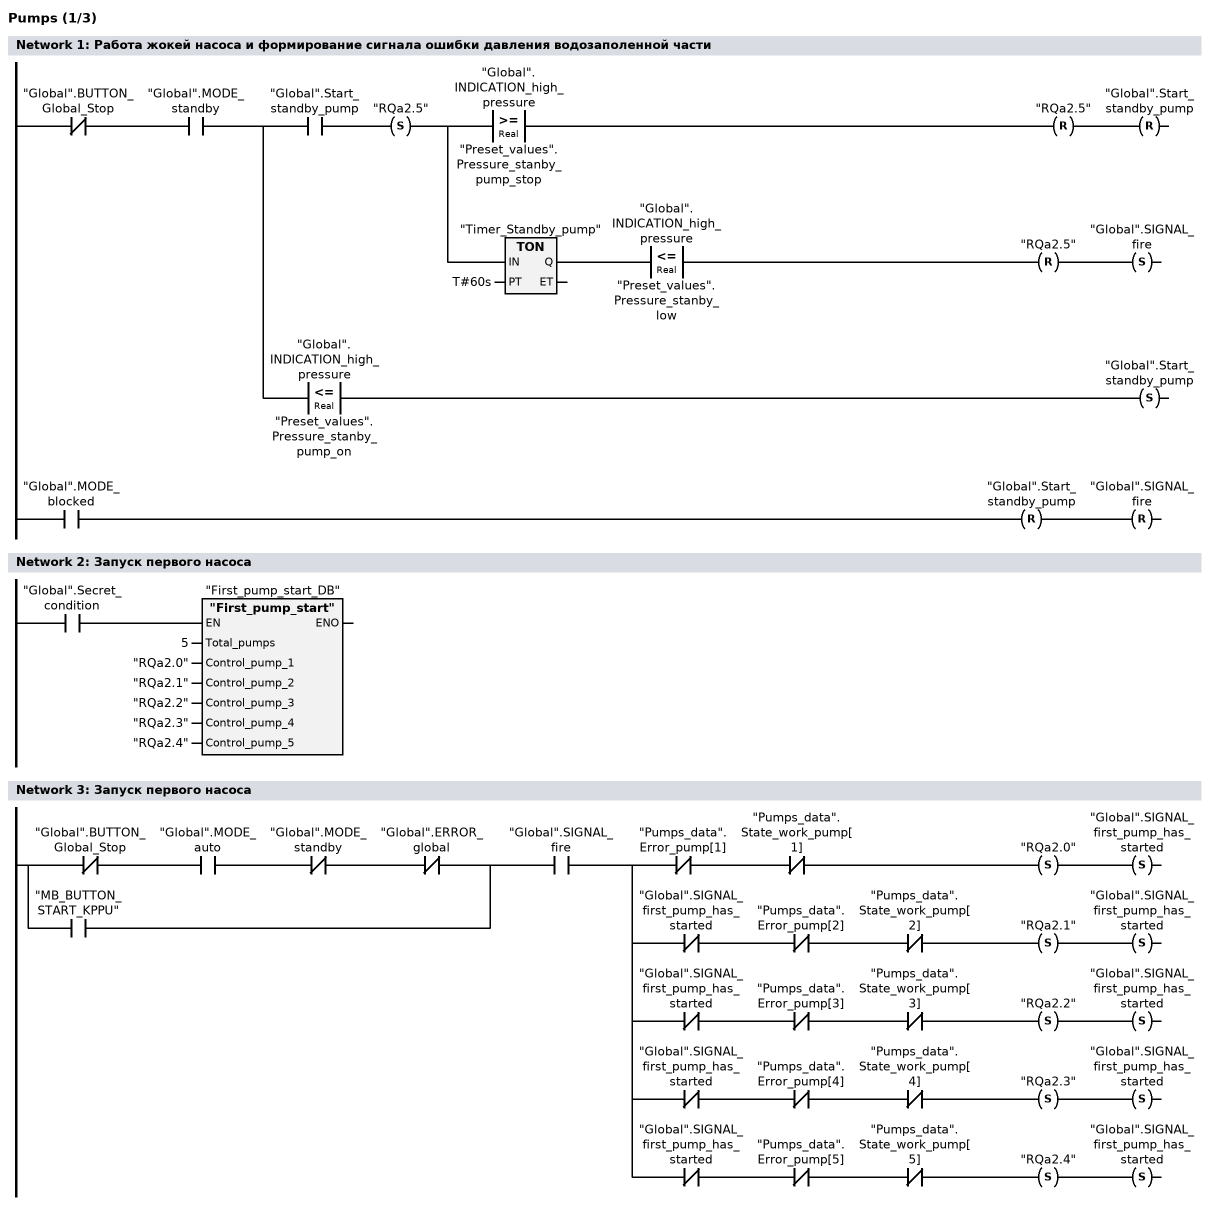
   #_w1 := NOT "Global".BUTTON_Global_Stop AND "Global".MODE_standby;
   #_w2 := #_w1 AND "Global".Start_standby_pump;
   IF #_w2 THEN "RQa2.5" := TRUE; END_IF;
   IF #_w2 AND ("Global".INDICATION_high_pressure >= "Preset_values".Pressure_stanby_pump_stop) THEN
       "RQa2.5" := FALSE;
       "Global".Start_standby_pump := FALSE;
   END_IF;
   "Timer_Standby_pump".TON(IN := #_w2, PT := T#60s);
   IF "Timer_Standby_pump".Q AND ("Global".INDICATION_high_pressure <= "Preset_values".Pressure_stanby_low) THEN
       "RQa2.5" := FALSE;
       "Global".SIGNAL_fire := TRUE;
   END_IF;
   IF #_w1 AND ("Global".INDICATION_high_pressure <= "Preset_values".Pressure_stanby_pump_on) THEN
       "Global".Start_standby_pump := TRUE;
   END_IF;
   IF "Global".MODE_blocked THEN
       "Global".Start_standby_pump := FALSE;
       "Global".SIGNAL_fire := FALSE;
   END_IF;
END_REGION

REGION Network 2: Запуск первого насоса
   RUNG wire#powerrail
      Contact( "Global".Secret_condition )
      "First_pump_start_DB"(Total_pumps := 5, Control_pump_1 := "RQa2.0", Control_pump_2 := "RQa2.1", Control_pump_3 := "RQa2.2", Control_pump_4 := "RQa2.3", Control_pump_5 := "RQa2.4")
   END_RUNG
   // the same network as SCL:
   IF "Global".Secret_condition THEN
       "First_pump_start_DB"(Total_pumps := 5,   // "First_pump_start"
                             Control_pump_1 := "RQa2.0",
                             Control_pump_2 := "RQa2.1",
                             Control_pump_3 := "RQa2.2",
                             Control_pump_4 := "RQa2.3",
                             Control_pump_5 := "RQa2.4");
   END_IF;
END_REGION

REGION Network 3: Запуск первого насоса
   RUNG wire#powerrail
      I_Contact( "Global".BUTTON_Global_Stop )
      Contact( "Global".MODE_auto )
      I_Contact( "Global".MODE_standby )
      I_Contact( "Global".ERROR_global )
      wire#w1
      Contact( "Global".SIGNAL_fire )
      wire#w2
      I_Contact( "Pumps_data".Error_pump[1] )
      I_Contact( "Pumps_data".State_work_pump[1] )
      S_Coil( "RQa2.0" )
      S_Coil( "Global".SIGNAL_first_pump_has_started )
   END_RUNG
   RUNG wire#powerrail
      Contact( "MB_BUTTON_START_KPPU" )
   END_RUNG wire#w1
   RUNG wire#w2
      I_Contact( "Global".SIGNAL_first_pump_has_started )
      I_Contact( "Pumps_data".Error_pump[2] )
      I_Contact( "Pumps_data".State_work_pump[2] )
      S_Coil( "RQa2.1" )
      S_Coil( "Global".SIGNAL_first_pump_has_started )
   END_RUNG
   RUNG wire#w2
      I_Contact( "Global".SIGNAL_first_pump_has_started )
      I_Contact( "Pumps_data".Error_pump[3] )
      I_Contact( "Pumps_data".State_work_pump[3] )
      S_Coil( "RQa2.2" )
      S_Coil( "Global".SIGNAL_first_pump_has_started )
   END_RUNG
   RUNG wire#w2
      I_Contact( "Global".SIGNAL_first_pump_has_started )
      I_Contact( "Pumps_data".Error_pump[4] )
      I_Contact( "Pumps_data".State_work_pump[4] )
      S_Coil( "RQa2.3" )
      S_Coil( "Global".SIGNAL_first_pump_has_started )
   END_RUNG
   RUNG wire#w2
      I_Contact( "Global".SIGNAL_first_pump_has_started )
      I_Contact( "Pumps_data".Error_pump[5] )
      I_Contact( "Pumps_data".State_work_pump[5] )
      S_Coil( "RQa2.4" )
      S_Coil( "Global".SIGNAL_first_pump_has_started )
   END_RUNG
   // the same network as SCL:
   #_w1 := ((NOT "Global".BUTTON_Global_Stop AND "Global".MODE_auto AND NOT "Global".MODE_standby AND NOT "Global".ERROR_global) OR "MB_BUTTON_START_KPPU") AND "Global".SIGNAL_fire;
   IF #_w1 AND NOT "Pumps_data".Error_pump[1] AND NOT "Pumps_data".State_work_pump[1] THEN
       "RQa2.0" := TRUE;
       "Global".SIGNAL_first_pump_has_started := TRUE;
   END_IF;
   IF #_w1 AND NOT "Global".SIGNAL_first_pump_has_started AND NOT "Pumps_data".Error_pump[2] AND NOT "Pumps_data".State_work_pump[2] THEN
       "RQa2.1" := TRUE;
       "Global".SIGNAL_first_pump_has_started := TRUE;
   END_IF;
   IF #_w1 AND NOT "Global".SIGNAL_first_pump_has_started AND NOT "Pumps_data".Error_pump[3] AND NOT "Pumps_data".State_work_pump[3] THEN
       "RQa2.2" := TRUE;
       "Global".SIGNAL_first_pump_has_started := TRUE;
   END_IF;
   IF #_w1 AND NOT "Global".SIGNAL_first_pump_has_started AND NOT "Pumps_data".Error_pump[4] AND NOT "Pumps_data".State_work_pump[4] THEN
       "RQa2.3" := TRUE;
       "Global".SIGNAL_first_pump_has_started := TRUE;
   END_IF;
   IF #_w1 AND NOT "Global".SIGNAL_first_pump_has_started AND NOT "Pumps_data".Error_pump[5] AND NOT "Pumps_data".State_work_pump[5] THEN
       "RQa2.4" := TRUE;
       "Global".SIGNAL_first_pump_has_started := TRUE;
   END_IF;
END_REGION

REGION Network 4: Каскадное включение/выключение насосов
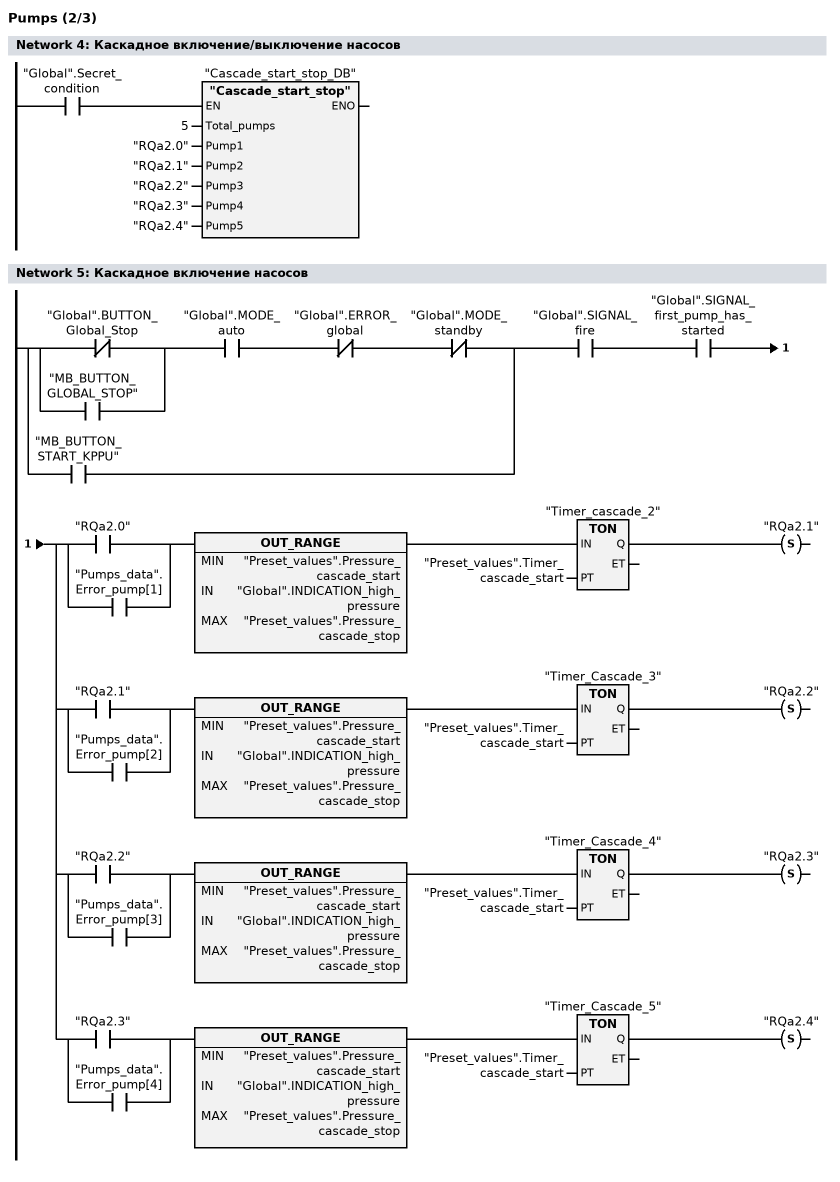
   RUNG wire#powerrail
      Contact( "Global".Secret_condition )
      "Cascade_start_stop_DB"(Total_pumps := 5, Pump1 := "RQa2.0", Pump2 := "RQa2.1", Pump3 := "RQa2.2", Pump4 := "RQa2.3", Pump5 := "RQa2.4")
   END_RUNG
   // the same network as SCL:
   IF "Global".Secret_condition THEN
       "Cascade_start_stop_DB"(Total_pumps := 5,   // "Cascade_start_stop"
                               Pump1 := "RQa2.0",
                               Pump2 := "RQa2.1",
                               Pump3 := "RQa2.2",
                               Pump4 := "RQa2.3",
                               Pump5 := "RQa2.4");
   END_IF;
END_REGION

REGION Network 5: Каскадное включение насосов
   #_w1 := (((NOT "Global".BUTTON_Global_Stop OR "MB_BUTTON_GLOBAL_STOP") AND "Global".MODE_auto AND NOT "Global".ERROR_global AND NOT "Global".MODE_standby) OR "MB_BUTTON_START_KPPU") AND "Global".SIGNAL_fire AND "Global".SIGNAL_first_pump_has_started;
   "Timer_cascade_2".TON(IN := #_w1 AND ("RQa2.0" OR "Pumps_data".Error_pump[1]) AND (("Global".INDICATION_high_pressure < "Preset_values".Pressure_cascade_start) OR ("Global".INDICATION_high_pressure > "Preset_values".Pressure_cascade_stop)),
                         PT := "Preset_values".Timer_cascade_start);
   IF "Timer_cascade_2".Q THEN "RQa2.1" := TRUE; END_IF;
   "Timer_Cascade_3".TON(IN := #_w1 AND ("RQa2.1" OR "Pumps_data".Error_pump[2]) AND (("Global".INDICATION_high_pressure < "Preset_values".Pressure_cascade_start) OR ("Global".INDICATION_high_pressure > "Preset_values".Pressure_cascade_stop)),
                         PT := "Preset_values".Timer_cascade_start);
   IF "Timer_Cascade_3".Q THEN "RQa2.2" := TRUE; END_IF;
   "Timer_Cascade_4".TON(IN := #_w1 AND ("RQa2.2" OR "Pumps_data".Error_pump[3]) AND (("Global".INDICATION_high_pressure < "Preset_values".Pressure_cascade_start) OR ("Global".INDICATION_high_pressure > "Preset_values".Pressure_cascade_stop)),
                         PT := "Preset_values".Timer_cascade_start);
   IF "Timer_Cascade_4".Q THEN "RQa2.3" := TRUE; END_IF;
   "Timer_Cascade_5".TON(IN := #_w1 AND ("RQa2.3" OR "Pumps_data".Error_pump[4]) AND (("Global".INDICATION_high_pressure < "Preset_values".Pressure_cascade_start) OR ("Global".INDICATION_high_pressure > "Preset_values".Pressure_cascade_stop)),
                         PT := "Preset_values".Timer_cascade_start);
   IF "Timer_Cascade_5".Q THEN "RQa2.4" := TRUE; END_IF;
END_REGION

REGION Network 6: Каскадное выключение насосов
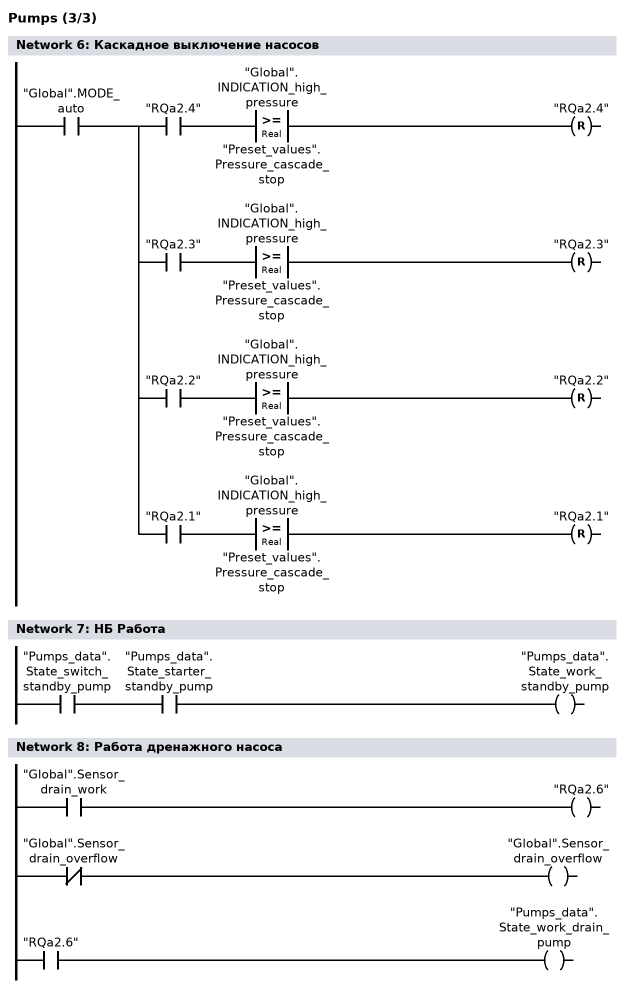
   RUNG wire#powerrail
      Contact( "Global".MODE_auto )
      wire#w1
      Contact( "RQa2.4" )
      { S7_Templates := "SrcType := Real" } GE_Contact(in1 := "Global".INDICATION_high_pressure, in2 := "Preset_values".Pressure_cascade_stop)
      R_Coil( "RQa2.4" )
   END_RUNG
   RUNG wire#w1
      Contact( "RQa2.3" )
      { S7_Templates := "SrcType := Real" } GE_Contact(in1 := "Global".INDICATION_high_pressure, in2 := "Preset_values".Pressure_cascade_stop)
      R_Coil( "RQa2.3" )
   END_RUNG
   RUNG wire#w1
      Contact( "RQa2.2" )
      { S7_Templates := "SrcType := Real" } GE_Contact(in1 := "Global".INDICATION_high_pressure, in2 := "Preset_values".Pressure_cascade_stop)
      R_Coil( "RQa2.2" )
   END_RUNG
   RUNG wire#w1
      Contact( "RQa2.1" )
      { S7_Templates := "SrcType := Real" } GE_Contact(in1 := "Global".INDICATION_high_pressure, in2 := "Preset_values".Pressure_cascade_stop)
      R_Coil( "RQa2.1" )
   END_RUNG
   // the same network as SCL:
   IF "Global".MODE_auto AND "RQa2.4" AND ("Global".INDICATION_high_pressure >= "Preset_values".Pressure_cascade_stop) THEN
       "RQa2.4" := FALSE;
   END_IF;
   IF "Global".MODE_auto AND "RQa2.3" AND ("Global".INDICATION_high_pressure >= "Preset_values".Pressure_cascade_stop) THEN
       "RQa2.3" := FALSE;
   END_IF;
   IF "Global".MODE_auto AND "RQa2.2" AND ("Global".INDICATION_high_pressure >= "Preset_values".Pressure_cascade_stop) THEN
       "RQa2.2" := FALSE;
   END_IF;
   IF "Global".MODE_auto AND "RQa2.1" AND ("Global".INDICATION_high_pressure >= "Preset_values".Pressure_cascade_stop) THEN
       "RQa2.1" := FALSE;
   END_IF;
END_REGION

REGION Network 7: НБ Работа
   RUNG wire#powerrail
      Contact( "Pumps_data".State_switch_standby_pump )
      Contact( "Pumps_data".State_starter_standby_pump )
      Coil( "Pumps_data".State_work_standby_pump )
   END_RUNG
   // the same network as SCL:
   "Pumps_data".State_work_standby_pump := "Pumps_data".State_switch_standby_pump AND "Pumps_data".State_starter_standby_pump;
END_REGION

REGION Network 8: Работа дренажного насоса
   RUNG wire#powerrail
      Contact( "Global".Sensor_drain_work )
      Coil( "RQa2.6" )
   END_RUNG
   RUNG wire#powerrail
      I_Contact( "Global".Sensor_drain_overflow )
      Coil( "Global".Sensor_drain_overflow )
   END_RUNG
   RUNG wire#powerrail
      Contact( "RQa2.6" )
      Coil( "Pumps_data".State_work_drain_pump )
   END_RUNG
   // the same network as SCL:
   "RQa2.6" := "Global".Sensor_drain_work;
   "Global".Sensor_drain_overflow := NOT "Global".Sensor_drain_overflow;
   "Pumps_data".State_work_drain_pump := "RQa2.6";
END_REGION
END_ORGANIZATION_BLOCK

ORGANIZATION_BLOCK "Modbus"   // OB127, LAD, ProgramCycle
TITLE = "Main Program Sweep (Cycle)"
{ S7_Optimized_Access := 'TRUE' }
VERSION : 0.1
   VAR_INPUT
      Initial_Call : Bool;   // Initial call of this OB
      Remanence : Bool;   // =True, if remanent data are available
   END_VAR
BEGIN

REGION Network 1
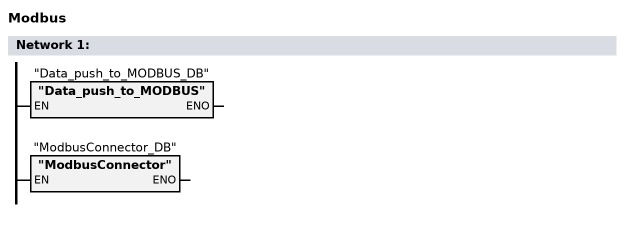
   RUNG wire#powerrail
      "Data_push_to_MODBUS_DB"()
   END_RUNG
   RUNG wire#powerrail
      "ModbusConnector_DB"()
   END_RUNG
   // the same network as SCL:
   "Data_push_to_MODBUS_DB"();   // "Data_push_to_MODBUS"
   "ModbusConnector_DB"();   // "ModbusConnector"
END_REGION
END_ORGANIZATION_BLOCK